Yaskawa INFORM job: A_ROOF_SIDE_0617_2_PAINT_45.JBI

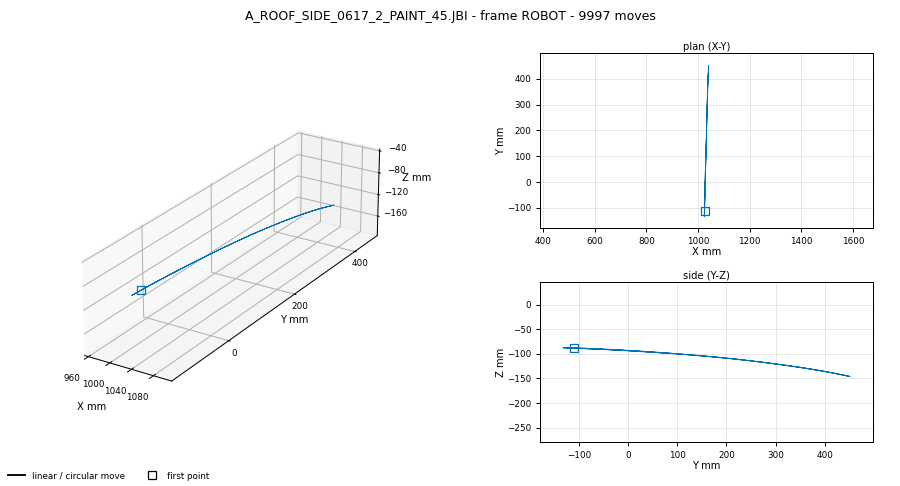
[picture p0: tool path of A_ROOF_SIDE_0617_2_PAINT_45.JBI in frame ROBOT, 9997 of 9997 moves have a stored position in this frame; points joined in program order, loops and branches not executed]
/JOB
//NAME A_ROOF_SIDE_0617_2_PAINT45
//POS
///NPOS 9997,0,0,0,0,0
///TOOL 1
///USER 0
///POSTYPE ROBOT
///RECTAN
///RCONF 1,0,0,0,0,0,0,0,0,0,0,0,0,0,0,0,0,0,0,0,0,0,0,0
C00000=1025.820,-110.808,-87.405,166.559,45.749,158.344
C00001=1025.826,-110.558,-87.414,166.562,45.746,158.343
C00002=1025.832,-110.309,-87.423,166.564,45.743,158.343
C00003=1025.837,-110.058,-87.432,166.568,45.740,158.343
C00004=1025.843,-109.809,-87.441,166.570,45.738,158.343
C00005=1025.849,-109.559,-87.450,166.574,45.735,158.343
C00006=1025.854,-109.310,-87.459,166.577,45.732,158.343
C00007=1025.860,-109.059,-87.468,166.579,45.729,158.343
C00008=1025.866,-108.810,-87.477,166.583,45.726,158.342
C00009=1025.872,-108.560,-87.486,166.586,45.724,158.342
C00010=1025.877,-108.311,-87.495,166.589,45.721,158.342
C00011=1025.883,-108.060,-87.504,166.592,45.718,158.342
C00012=1025.889,-107.811,-87.513,166.594,45.716,158.342
C00013=1025.895,-107.561,-87.522,166.598,45.713,158.342
C00014=1025.900,-107.312,-87.531,166.601,45.710,158.342
C00015=1025.906,-107.061,-87.540,166.604,45.708,158.341
C00016=1025.912,-106.812,-87.550,166.607,45.705,158.341
C00017=1025.918,-106.562,-87.558,166.609,45.703,158.341
C00018=1025.924,-106.312,-87.568,166.613,45.700,158.341
C00019=1025.929,-106.063,-87.577,166.616,45.697,158.341
C00020=1025.935,-105.812,-87.586,166.618,45.694,158.341
C00021=1025.941,-105.563,-87.595,166.622,45.692,158.341
C00022=1025.946,-105.313,-87.605,166.624,45.689,158.340
C00023=1025.952,-105.063,-87.614,166.628,45.686,158.340
C00024=1025.958,-104.814,-87.623,166.630,45.684,158.340
C00025=1025.964,-104.564,-87.633,166.634,45.681,158.340
C00026=1025.969,-104.314,-87.641,166.637,45.678,158.340
C00027=1025.975,-104.064,-87.651,166.640,45.676,158.340
C00028=1025.981,-103.814,-87.661,166.643,45.673,158.340
C00029=1025.986,-103.565,-87.670,166.645,45.670,158.340
C00030=1025.992,-103.315,-87.679,166.649,45.668,158.340
C00031=1025.998,-103.066,-87.688,166.651,45.665,158.339
C00032=1026.004,-102.816,-87.698,166.654,45.662,158.339
C00033=1026.010,-102.566,-87.707,166.658,45.659,158.339
C00034=1026.014,-102.316,-87.717,166.660,45.657,158.339
C00035=1026.021,-102.066,-87.726,166.664,45.654,158.339
C00036=1026.027,-101.817,-87.736,166.666,45.652,158.339
C00037=1026.032,-101.567,-87.745,166.670,45.649,158.339
C00038=1026.039,-101.281,-87.756,166.673,45.646,158.338
C00039=1026.046,-100.994,-87.767,166.676,45.643,158.338
C00040=1026.052,-100.708,-87.777,166.679,45.640,158.338
C00041=1026.059,-100.422,-87.789,166.683,45.637,158.338
C00042=1026.064,-100.173,-87.797,166.686,45.634,158.338
C00043=1026.070,-99.923,-87.807,166.690,45.631,158.338
C00044=1026.077,-99.673,-87.816,166.692,45.629,158.337
C00045=1026.083,-99.423,-87.826,166.696,45.626,158.337
C00046=1026.088,-99.174,-87.836,166.698,45.624,158.337
C00047=1026.094,-98.924,-87.845,166.701,45.621,158.337
C00048=1026.100,-98.674,-87.855,166.704,45.619,158.337
C00049=1026.106,-98.424,-87.864,166.707,45.616,158.337
C00050=1026.111,-98.175,-87.873,166.711,45.613,158.337
C00051=1026.117,-97.925,-87.883,166.713,45.610,158.336
C00052=1026.123,-97.675,-87.893,166.716,45.608,158.336
C00053=1026.129,-97.425,-87.902,166.719,45.605,158.336
C00054=1026.134,-97.176,-87.912,166.722,45.603,158.336
C00055=1026.140,-96.926,-87.922,166.725,45.600,158.336
C00056=1026.146,-96.676,-87.932,166.728,45.598,158.336
C00057=1026.152,-96.426,-87.941,166.731,45.595,158.336
C00058=1026.157,-96.176,-87.951,166.734,45.593,158.336
C00059=1026.163,-95.927,-87.961,166.737,45.590,158.336
C00060=1026.168,-95.677,-87.972,166.740,45.588,158.336
C00061=1026.175,-95.427,-87.981,166.742,45.585,158.335
C00062=1026.179,-95.178,-87.991,166.746,45.583,158.335
C00063=1026.186,-94.928,-88.001,166.748,45.580,158.335
C00064=1026.192,-94.678,-88.010,166.752,45.577,158.335
C00065=1026.197,-94.428,-88.020,166.754,45.575,158.335
C00066=1026.203,-94.178,-88.030,166.758,45.572,158.335
C00067=1026.208,-93.929,-88.040,166.760,45.570,158.335
C00068=1026.214,-93.679,-88.049,166.764,45.567,158.334
C00069=1026.220,-93.430,-88.060,166.766,45.565,158.334
C00070=1026.226,-93.180,-88.070,166.770,45.562,158.334
C00071=1026.232,-92.930,-88.080,166.772,45.560,158.334
C00072=1026.238,-92.680,-88.089,166.775,45.557,158.334
C00073=1026.243,-92.431,-88.099,166.778,45.555,158.334
C00074=1026.249,-92.182,-88.109,166.781,45.552,158.334
C00075=1026.255,-91.931,-88.120,166.785,45.550,158.334
C00076=1026.261,-91.682,-88.129,166.787,45.547,158.334
C00077=1026.266,-91.431,-88.139,166.791,45.545,158.334
C00078=1026.272,-91.182,-88.149,166.793,45.542,158.333
C00079=1026.278,-90.932,-88.160,166.797,45.539,158.333
C00080=1026.284,-90.682,-88.169,166.799,45.537,158.333
C00081=1026.289,-90.433,-88.179,166.802,45.534,158.333
C00082=1026.295,-90.183,-88.189,166.805,45.532,158.333
C00083=1026.301,-89.934,-88.200,166.808,45.529,158.333
C00084=1026.307,-89.684,-88.209,166.811,45.527,158.333
C00085=1026.313,-89.434,-88.219,166.814,45.524,158.332
C00086=1026.319,-89.185,-88.230,166.817,45.522,158.332
C00087=1026.325,-88.935,-88.240,166.820,45.519,158.332
C00088=1026.331,-88.685,-88.249,166.823,45.516,158.332
C00089=1026.336,-88.435,-88.260,166.826,45.514,158.332
C00090=1026.343,-88.185,-88.270,166.828,45.512,158.332
C00091=1026.348,-87.935,-88.280,166.832,45.509,158.332
C00092=1026.354,-87.686,-88.290,166.834,45.507,158.332
C00093=1026.360,-87.436,-88.300,166.838,45.504,158.332
C00094=1026.366,-87.186,-88.310,166.840,45.502,158.331
C00095=1026.372,-86.937,-88.321,166.844,45.499,158.331
C00096=1026.377,-86.687,-88.331,166.846,45.497,158.331
C00097=1026.384,-86.437,-88.341,166.850,45.494,158.331
C00098=1026.389,-86.187,-88.351,166.852,45.492,158.331
C00099=1026.395,-85.938,-88.361,166.856,45.489,158.331
C00100=1026.401,-85.688,-88.372,166.858,45.487,158.331
C00101=1026.407,-85.438,-88.381,166.861,45.484,158.330
C00102=1026.414,-85.154,-88.393,166.865,45.481,158.330
C00103=1026.420,-84.871,-88.404,166.868,45.478,158.330
C00104=1026.427,-84.586,-88.416,166.871,45.475,158.330
C00105=1026.434,-84.303,-88.428,166.875,45.472,158.330
C00106=1026.440,-84.053,-88.438,166.877,45.470,158.330
C00107=1026.445,-83.803,-88.449,166.881,45.467,158.330
C00108=1026.452,-83.554,-88.458,166.884,45.465,158.330
C00109=1026.458,-83.303,-88.469,166.887,45.462,158.329
C00110=1026.464,-83.054,-88.479,166.890,45.459,158.329
C00111=1026.470,-82.804,-88.490,166.893,45.457,158.329
C00112=1026.476,-82.554,-88.499,166.896,45.454,158.329
C00113=1026.482,-82.305,-88.510,166.899,45.452,158.329
C00114=1026.488,-82.055,-88.520,166.902,45.449,158.329
C00115=1026.494,-81.806,-88.531,166.904,45.446,158.328
C00116=1026.499,-81.556,-88.541,166.908,45.444,158.328
C00117=1026.506,-81.306,-88.551,166.910,45.441,158.328
C00118=1026.511,-81.056,-88.561,166.914,45.439,158.328
C00119=1026.518,-80.806,-88.572,166.916,45.436,158.328
C00120=1026.524,-80.557,-88.583,166.919,45.433,158.328
C00121=1026.530,-80.307,-88.592,166.922,45.431,158.328
C00122=1026.536,-80.058,-88.603,166.925,45.428,158.328
C00123=1026.541,-79.807,-88.614,166.928,45.426,158.327
C00124=1026.547,-79.558,-88.624,166.931,45.424,158.327
C00125=1026.553,-79.309,-88.635,166.934,45.421,158.327
C00126=1026.559,-79.058,-88.645,166.937,45.419,158.327
C00127=1026.565,-78.808,-88.656,166.940,45.417,158.327
C00128=1026.571,-78.559,-88.667,166.943,45.414,158.327
C00129=1026.577,-78.310,-88.678,166.946,45.412,158.327
C00130=1026.582,-78.059,-88.688,166.948,45.410,158.327
C00131=1026.589,-77.810,-88.698,166.952,45.407,158.326
C00132=1026.595,-77.560,-88.710,166.954,45.405,158.326
C00133=1026.601,-77.311,-88.720,166.958,45.402,158.326
C00134=1026.606,-77.061,-88.731,166.960,45.400,158.326
C00135=1026.612,-76.811,-88.741,166.963,45.397,158.326
C00136=1026.618,-76.561,-88.752,166.966,45.395,158.326
C00137=1026.624,-76.312,-88.763,166.970,45.392,158.326
C00138=1026.630,-76.062,-88.774,166.972,45.390,158.326
C00139=1026.636,-75.813,-88.785,166.976,45.387,158.326
C00140=1026.642,-75.562,-88.795,166.978,45.385,158.325
C00141=1026.647,-75.313,-88.806,166.980,45.383,158.325
C00142=1026.653,-75.064,-88.817,166.984,45.380,158.325
C00143=1026.660,-74.814,-88.827,166.986,45.378,158.325
C00144=1026.666,-74.564,-88.838,166.990,45.375,158.325
C00145=1026.672,-74.315,-88.849,166.992,45.373,158.325
C00146=1026.677,-74.065,-88.860,166.996,45.371,158.325
C00147=1026.684,-73.815,-88.871,166.998,45.368,158.325
C00148=1026.689,-73.565,-88.881,167.001,45.366,158.324
C00149=1026.694,-73.315,-88.893,167.004,45.364,158.324
C00150=1026.700,-73.066,-88.904,167.007,45.362,158.324
C00151=1026.706,-72.815,-88.915,167.009,45.359,158.324
C00152=1026.712,-72.566,-88.926,167.013,45.357,158.324
C00153=1026.718,-72.316,-88.937,167.016,45.355,158.324
C00154=1026.724,-72.068,-88.948,167.019,45.352,158.324
C00155=1026.730,-71.817,-88.960,167.021,45.350,158.324
C00156=1026.736,-71.568,-88.970,167.024,45.348,158.324
C00157=1026.741,-71.318,-88.982,167.028,45.345,158.324
C00158=1026.747,-71.068,-88.993,167.030,45.343,158.323
C00159=1026.753,-70.818,-89.004,167.033,45.341,158.323
C00160=1026.759,-70.569,-89.015,167.036,45.338,158.323
C00161=1026.764,-70.319,-89.026,167.039,45.336,158.323
C00162=1026.771,-70.069,-89.037,167.042,45.333,158.323
C00163=1026.776,-69.820,-89.048,167.045,45.331,158.323
C00164=1026.782,-69.570,-89.059,167.047,45.329,158.323
C00165=1026.788,-69.320,-89.071,167.051,45.326,158.323
C00166=1026.795,-69.039,-89.083,167.054,45.324,158.323
C00167=1026.801,-68.757,-89.096,167.056,45.322,158.323
C00168=1026.808,-68.475,-89.108,167.060,45.319,158.322
C00169=1026.814,-68.193,-89.121,167.063,45.316,158.322
C00170=1026.821,-67.944,-89.133,167.066,45.314,158.322
///RCONF 1,0,0,1,0,0,0,0,0,0,0,0,0,0,0,0,0,0,0,0,0,0,0,0
C00171=1026.827,-67.694,-89.143,167.069,45.311,158.322
C00172=1026.832,-67.445,-89.154,167.072,45.309,158.322
C00173=1026.838,-67.194,-89.166,167.075,45.307,158.322
C00174=1026.844,-66.945,-89.177,167.078,45.305,158.322
C00175=1026.850,-66.695,-89.189,167.080,45.302,158.322
C00176=1026.856,-66.445,-89.200,167.084,45.300,158.322
C00177=1026.862,-66.196,-89.211,167.087,45.298,158.322
C00178=1026.868,-65.946,-89.222,167.089,45.296,158.321
C00179=1026.874,-65.697,-89.234,167.093,45.293,158.321
C00180=1026.880,-65.446,-89.245,167.095,45.291,158.321
C00181=1026.885,-65.197,-89.256,167.097,45.289,158.321
C00182=1026.891,-64.947,-89.267,167.101,45.286,158.321
C00183=1026.898,-64.698,-89.279,167.104,45.284,158.321
C00184=1026.904,-64.448,-89.290,167.107,45.281,158.321
C00185=1026.910,-64.198,-89.301,167.110,45.279,158.321
C00186=1026.915,-63.949,-89.313,167.112,45.277,158.320
C00187=1026.922,-63.699,-89.325,167.116,45.274,158.320
C00188=1026.927,-63.449,-89.336,167.118,45.272,158.320
C00189=1026.933,-63.200,-89.347,167.121,45.270,158.320
C00190=1026.940,-62.950,-89.358,167.124,45.268,158.320
C00191=1026.945,-62.700,-89.370,167.127,45.266,158.320
C00192=1026.951,-62.451,-89.382,167.130,45.263,158.320
C00193=1026.957,-62.201,-89.393,167.133,45.261,158.320
C00194=1026.963,-61.951,-89.404,167.135,45.259,158.320
C00195=1026.969,-61.702,-89.416,167.138,45.256,158.319
C00196=1026.976,-61.452,-89.427,167.141,45.254,158.319
C00197=1026.981,-61.202,-89.438,167.144,45.252,158.319
C00198=1026.987,-60.953,-89.450,167.147,45.249,158.319
C00199=1026.993,-60.703,-89.461,167.150,45.247,158.319
C00200=1027.000,-60.454,-89.473,167.152,45.245,158.319
C00201=1027.006,-60.204,-89.484,167.156,45.242,158.319
C00202=1027.011,-59.954,-89.497,167.158,45.240,158.319
C00203=1027.018,-59.704,-89.508,167.162,45.238,158.319
C00204=1027.024,-59.455,-89.519,167.164,45.235,158.318
C00205=1027.030,-59.205,-89.531,167.167,45.233,158.318
C00206=1027.036,-58.956,-89.541,167.170,45.230,158.318
C00207=1027.042,-58.706,-89.554,167.173,45.228,158.318
C00208=1027.048,-58.456,-89.565,167.175,45.226,158.318
C00209=1027.054,-58.207,-89.577,167.178,45.223,158.318
C00210=1027.061,-57.956,-89.588,167.181,45.221,158.318
C00211=1027.066,-57.707,-89.600,167.185,45.219,158.318
C00212=1027.072,-57.457,-89.612,167.187,45.216,158.317
C00213=1027.078,-57.208,-89.623,167.190,45.214,158.317
C00214=1027.085,-56.958,-89.634,167.193,45.211,158.317
C00215=1027.091,-56.708,-89.646,167.195,45.209,158.317
C00216=1027.097,-56.459,-89.659,167.198,45.207,158.317
C00217=1027.103,-56.209,-89.670,167.201,45.204,158.317
C00218=1027.109,-55.960,-89.681,167.204,45.202,158.317
C00219=1027.115,-55.710,-89.693,167.207,45.199,158.316
C00220=1027.122,-55.460,-89.705,167.210,45.197,158.316
C00221=1027.127,-55.211,-89.716,167.213,45.195,158.316
C00222=1027.134,-54.961,-89.728,167.216,45.192,158.316
C00223=1027.140,-54.712,-89.740,167.218,45.190,158.316
C00224=1027.146,-54.462,-89.751,167.221,45.188,158.316
C00225=1027.152,-54.212,-89.763,167.224,45.185,158.316
C00226=1027.158,-53.962,-89.775,167.227,45.183,158.316
C00227=1027.164,-53.713,-89.786,167.229,45.181,158.315
C00228=1027.171,-53.464,-89.798,167.233,45.179,158.315
C00229=1027.177,-53.213,-89.810,167.235,45.176,158.315
C00230=1027.183,-52.933,-89.823,167.239,45.174,158.315
C00231=1027.191,-52.652,-89.836,167.242,45.171,158.315
C00232=1027.197,-52.372,-89.850,167.246,45.168,158.315
C00233=1027.205,-52.091,-89.863,167.248,45.165,158.315
C00234=1027.211,-51.842,-89.874,167.252,45.163,158.314
C00235=1027.217,-51.592,-89.886,167.254,45.160,158.314
C00236=1027.223,-51.342,-89.899,167.256,45.158,158.314
C00237=1027.230,-51.092,-89.910,167.260,45.156,158.314
C00238=1027.236,-50.843,-89.922,167.262,45.153,158.314
C00239=1027.241,-50.593,-89.934,167.266,45.151,158.314
C00240=1027.248,-50.344,-89.946,167.269,45.149,158.314
C00241=1027.254,-50.093,-89.958,167.271,45.146,158.314
C00242=1027.259,-49.844,-89.970,167.273,45.144,158.313
C00243=1027.266,-49.594,-89.982,167.277,45.142,158.313
C00244=1027.272,-49.345,-89.995,167.280,45.140,158.313
C00245=1027.278,-49.095,-90.007,167.282,45.138,158.313
C00246=1027.284,-48.846,-90.019,167.285,45.136,158.313
C00247=1027.289,-48.596,-90.031,167.288,45.133,158.313
C00248=1027.296,-48.346,-90.043,167.291,45.131,158.313
C00249=1027.302,-48.096,-90.056,167.293,45.129,158.313
C00250=1027.308,-47.848,-90.067,167.296,45.127,158.313
C00251=1027.314,-47.598,-90.080,167.299,45.125,158.313
C00252=1027.320,-47.348,-90.093,167.302,45.122,158.312
C00253=1027.326,-47.098,-90.105,167.304,45.120,158.312
C00254=1027.332,-46.849,-90.117,167.307,45.118,158.312
C00255=1027.338,-46.599,-90.129,167.311,45.116,158.312
C00256=1027.344,-46.350,-90.141,167.313,45.113,158.312
C00257=1027.350,-46.100,-90.154,167.316,45.111,158.312
C00258=1027.356,-45.850,-90.166,167.319,45.109,158.312
C00259=1027.362,-45.601,-90.178,167.322,45.107,158.312
C00260=1027.368,-45.351,-90.191,167.324,45.105,158.312
C00261=1027.375,-45.102,-90.202,167.327,45.103,158.311
C00262=1027.381,-44.852,-90.215,167.330,45.100,158.311
C00263=1027.387,-44.602,-90.228,167.333,45.098,158.311
C00264=1027.393,-44.352,-90.240,167.335,45.096,158.311
C00265=1027.399,-44.103,-90.252,167.338,45.094,158.311
C00266=1027.404,-43.853,-90.264,167.341,45.091,158.311
C00267=1027.411,-43.604,-90.276,167.344,45.089,158.311
C00268=1027.417,-43.354,-90.289,167.346,45.087,158.311
C00269=1027.423,-43.104,-90.301,167.349,45.085,158.310
C00270=1027.430,-42.854,-90.313,167.352,45.083,158.310
C00271=1027.436,-42.605,-90.327,167.355,45.081,158.310
C00272=1027.441,-42.356,-90.339,167.358,45.079,158.310
C00273=1027.448,-42.106,-90.351,167.360,45.076,158.310
C00274=1027.454,-41.856,-90.363,167.364,45.074,158.310
C00275=1027.460,-41.606,-90.376,167.366,45.072,158.310
C00276=1027.466,-41.357,-90.388,167.369,45.070,158.310
C00277=1027.472,-41.107,-90.400,167.371,45.067,158.309
C00278=1027.478,-40.858,-90.414,167.375,45.065,158.309
C00279=1027.485,-40.608,-90.426,167.377,45.063,158.309
C00280=1027.491,-40.358,-90.438,167.380,45.061,158.309
C00281=1027.497,-40.108,-90.451,167.382,45.058,158.309
C00282=1027.503,-39.859,-90.463,167.386,45.056,158.309
C00283=1027.509,-39.610,-90.476,167.388,45.054,158.309
C00284=1027.515,-39.360,-90.488,167.391,45.051,158.309
C00285=1027.522,-39.111,-90.500,167.394,45.049,158.309
C00286=1027.528,-38.861,-90.513,167.397,45.047,158.308
C00287=1027.534,-38.612,-90.526,167.399,45.045,158.308
C00288=1027.540,-38.362,-90.538,167.402,45.043,158.308
C00289=1027.546,-38.112,-90.551,167.405,45.041,158.308
C00290=1027.551,-37.862,-90.564,167.408,45.038,158.308
C00291=1027.558,-37.613,-90.577,167.411,45.036,158.308
C00292=1027.564,-37.363,-90.589,167.413,45.034,158.308
C00293=1027.570,-37.114,-90.603,167.416,45.032,158.308
C00294=1027.577,-36.833,-90.617,167.419,45.030,158.308
C00295=1027.584,-36.553,-90.631,167.422,45.027,158.307
C00296=1027.590,-36.273,-90.645,167.425,45.025,158.307
C00297=1027.597,-35.993,-90.660,167.428,45.023,158.307
C00298=1027.603,-35.743,-90.673,167.431,45.020,158.307
C00299=1027.610,-35.494,-90.685,167.434,45.018,158.307
C00300=1027.616,-35.244,-90.698,167.436,45.016,158.307
C00301=1027.622,-34.994,-90.710,167.439,45.014,158.307
C00302=1027.628,-34.745,-90.724,167.442,45.012,158.307
C00303=1027.634,-34.495,-90.736,167.445,45.010,158.307
C00304=1027.640,-34.246,-90.749,167.447,45.007,158.306
C00305=1027.646,-33.996,-90.762,167.450,45.005,158.306
C00306=1027.652,-33.747,-90.775,167.453,45.003,158.306
C00307=1027.658,-33.497,-90.788,167.455,45.001,158.306
C00308=1027.664,-33.247,-90.801,167.458,44.999,158.306
C00309=1027.670,-32.998,-90.814,167.461,44.997,158.306
C00310=1027.676,-32.748,-90.827,167.464,44.995,158.306
C00311=1027.682,-32.498,-90.839,167.466,44.993,158.306
C00312=1027.688,-32.249,-90.853,167.469,44.991,158.306
C00313=1027.695,-31.999,-90.866,167.471,44.989,158.305
C00314=1027.701,-31.749,-90.879,167.475,44.986,158.305
C00315=1027.707,-31.499,-90.891,167.477,44.984,158.305
C00316=1027.713,-31.250,-90.905,167.480,44.982,158.305
C00317=1027.719,-31.001,-90.918,167.483,44.980,158.305
C00318=1027.726,-30.751,-90.930,167.485,44.978,158.305
C00319=1027.732,-30.502,-90.943,167.489,44.976,158.305
C00320=1027.738,-30.252,-90.956,167.491,44.973,158.305
C00321=1027.744,-30.003,-90.969,167.494,44.971,158.304
C00322=1027.750,-29.753,-90.982,167.496,44.969,158.304
C00323=1027.757,-29.503,-90.995,167.499,44.967,158.304
C00324=1027.763,-29.254,-91.008,167.501,44.965,158.304
C00325=1027.769,-29.004,-91.021,167.505,44.962,158.304
C00326=1027.775,-28.755,-91.034,167.507,44.960,158.304
C00327=1027.782,-28.505,-91.048,167.510,44.958,158.304
C00328=1027.788,-28.255,-91.060,167.513,44.956,158.304
C00329=1027.794,-28.006,-91.073,167.515,44.953,158.303
C00330=1027.801,-27.756,-91.087,167.518,44.951,158.303
C00331=1027.806,-27.506,-91.100,167.521,44.949,158.303
C00332=1027.813,-27.257,-91.113,167.524,44.947,158.303
C00333=1027.819,-27.008,-91.126,167.526,44.945,158.303
C00334=1027.824,-26.758,-91.139,167.529,44.943,158.303
C00335=1027.830,-26.508,-91.153,167.531,44.941,158.303
C00336=1027.837,-26.258,-91.166,167.534,44.939,158.303
C00337=1027.843,-26.009,-91.179,167.536,44.937,158.303
C00338=1027.849,-25.760,-91.193,167.540,44.934,158.302
C00339=1027.855,-25.510,-91.206,167.543,44.932,158.302
C00340=1027.861,-25.260,-91.219,167.545,44.930,158.302
///RCONF 1,0,0,0,0,0,0,0,0,0,0,0,0,0,0,0,0,0,0,0,0,0,0,0
C00341=1027.867,-25.011,-91.232,167.548,44.928,158.302
C00342=1027.873,-24.761,-91.247,167.550,44.926,158.302
C00343=1027.879,-24.512,-91.260,167.553,44.925,158.302
C00344=1027.886,-24.262,-91.273,167.555,44.923,158.302
C00345=1027.892,-24.012,-91.286,167.558,44.921,158.302
C00346=1027.897,-23.763,-91.300,167.561,44.919,158.302
C00347=1027.904,-23.513,-91.313,167.564,44.916,158.302
C00348=1027.910,-23.264,-91.326,167.567,44.914,158.301
C00349=1027.916,-23.014,-91.340,167.569,44.912,158.301
C00350=1027.922,-22.765,-91.354,167.572,44.910,158.301
C00351=1027.928,-22.516,-91.367,167.574,44.908,158.301
C00352=1027.935,-22.266,-91.381,167.577,44.906,158.301
C00353=1027.941,-22.016,-91.394,167.579,44.904,158.301
C00354=1027.946,-21.767,-91.408,167.582,44.902,158.301
C00355=1027.953,-21.518,-91.421,167.585,44.900,158.301
C00356=1027.959,-21.267,-91.434,167.588,44.898,158.301
C00357=1027.965,-21.018,-91.447,167.591,44.895,158.300
C00358=1027.972,-20.737,-91.463,167.593,44.893,158.300
C00359=1027.979,-20.455,-91.479,167.597,44.891,158.300
C00360=1027.986,-20.175,-91.493,167.599,44.888,158.300
C00361=1027.993,-19.894,-91.508,167.603,44.886,158.300
C00362=1027.999,-19.644,-91.522,167.605,44.884,158.300
C00363=1028.006,-19.394,-91.535,167.608,44.881,158.300
C00364=1028.011,-19.145,-91.549,167.610,44.879,158.299
C00365=1028.018,-18.896,-91.562,167.613,44.877,158.299
C00366=1028.024,-18.646,-91.576,167.615,44.875,158.299
C00367=1028.030,-18.396,-91.590,167.618,44.873,158.299
C00368=1028.036,-18.147,-91.603,167.622,44.871,158.299
C00369=1028.043,-17.897,-91.617,167.624,44.869,158.299
C00370=1028.049,-17.648,-91.630,167.627,44.867,158.299
C00371=1028.055,-17.398,-91.644,167.629,44.865,158.299
C00372=1028.061,-17.148,-91.658,167.632,44.863,158.298
C00373=1028.068,-16.899,-91.672,167.634,44.861,158.298
C00374=1028.073,-16.650,-91.685,167.637,44.859,158.298
C00375=1028.080,-16.400,-91.699,167.639,44.856,158.298
C00376=1028.087,-16.151,-91.712,167.642,44.854,158.298
C00377=1028.093,-15.901,-91.726,167.645,44.852,158.298
C00378=1028.099,-15.651,-91.740,167.648,44.850,158.298
C00379=1028.105,-15.402,-91.753,167.651,44.848,158.298
C00380=1028.111,-15.151,-91.767,167.653,44.846,158.298
C00381=1028.118,-14.903,-91.781,167.656,44.844,158.297
C00382=1028.123,-14.653,-91.795,167.658,44.842,158.297
C00383=1028.130,-14.403,-91.809,167.661,44.840,158.297
C00384=1028.135,-14.154,-91.823,167.663,44.838,158.297
C00385=1028.142,-13.904,-91.836,167.666,44.836,158.297
C00386=1028.148,-13.655,-91.851,167.669,44.834,158.297
C00387=1028.153,-13.405,-91.865,167.671,44.832,158.297
C00388=1028.160,-13.155,-91.878,167.674,44.829,158.297
C00389=1028.166,-12.906,-91.893,167.676,44.827,158.296
C00390=1028.172,-12.657,-91.906,167.679,44.825,158.296
C00391=1028.178,-12.407,-91.921,167.681,44.824,158.296
C00392=1028.185,-12.157,-91.934,167.684,44.822,158.296
C00393=1028.191,-11.908,-91.949,167.687,44.820,158.296
C00394=1028.197,-11.659,-91.962,167.689,44.818,158.296
C00395=1028.203,-11.408,-91.976,167.692,44.816,158.296
C00396=1028.210,-11.160,-91.990,167.694,44.814,158.296
C00397=1028.215,-10.910,-92.004,167.697,44.812,158.296
C00398=1028.221,-10.660,-92.018,167.699,44.810,158.295
C00399=1028.228,-10.411,-92.032,167.703,44.808,158.295
C00400=1028.234,-10.161,-92.047,167.706,44.806,158.295
C00401=1028.240,-9.912,-92.061,167.708,44.804,158.295
C00402=1028.247,-9.662,-92.075,167.711,44.801,158.295
C00403=1028.253,-9.413,-92.088,167.713,44.799,158.295
C00404=1028.259,-9.163,-92.103,167.716,44.797,158.295
C00405=1028.265,-8.913,-92.117,167.718,44.795,158.295
C00406=1028.271,-8.663,-92.130,167.721,44.793,158.295
C00407=1028.277,-8.415,-92.145,167.723,44.791,158.294
C00408=1028.284,-8.165,-92.159,167.726,44.789,158.294
C00409=1028.290,-7.916,-92.173,167.729,44.787,158.294
C00410=1028.297,-7.666,-92.187,167.731,44.785,158.294
C00411=1028.302,-7.417,-92.201,167.734,44.783,158.294
C00412=1028.308,-7.166,-92.216,167.736,44.781,158.294
C00413=1028.315,-6.918,-92.230,167.739,44.779,158.294
C00414=1028.321,-6.667,-92.244,167.741,44.777,158.294
C00415=1028.327,-6.418,-92.257,167.744,44.775,158.293
C00416=1028.334,-6.169,-92.272,167.747,44.773,158.293
C00417=1028.340,-5.919,-92.285,167.749,44.771,158.293
C00418=1028.346,-5.670,-92.300,167.751,44.768,158.293
C00419=1028.352,-5.420,-92.314,167.754,44.766,158.293
C00420=1028.359,-5.171,-92.329,167.757,44.764,158.293
C00421=1028.364,-4.921,-92.342,167.759,44.762,158.293
C00422=1028.372,-4.639,-92.359,167.763,44.760,158.293
C00423=1028.379,-4.356,-92.375,167.765,44.757,158.292
C00424=1028.386,-4.072,-92.391,167.769,44.755,158.292
C00425=1028.394,-3.791,-92.407,167.771,44.752,158.292
C00426=1028.399,-3.542,-92.422,167.774,44.751,158.292
C00427=1028.405,-3.291,-92.436,167.776,44.749,158.292
C00428=1028.412,-3.042,-92.451,167.779,44.747,158.292
C00429=1028.418,-2.793,-92.466,167.782,44.745,158.292
C00430=1028.424,-2.542,-92.480,167.784,44.743,158.292
C00431=1028.429,-2.293,-92.494,167.787,44.741,158.291
C00432=1028.436,-2.044,-92.509,167.789,44.739,158.291
C00433=1028.441,-1.794,-92.523,167.792,44.737,158.291
C00434=1028.448,-1.545,-92.538,167.795,44.735,158.291
C00435=1028.454,-1.296,-92.552,167.797,44.734,158.291
C00436=1028.461,-1.046,-92.567,167.800,44.732,158.291
C00437=1028.467,-0.796,-92.581,167.802,44.730,158.291
C00438=1028.472,-0.547,-92.596,167.805,44.728,158.291
C00439=1028.479,-0.297,-92.611,167.808,44.726,158.291
C00440=1028.485,-0.048,-92.626,167.810,44.724,158.290
C00441=1028.491,0.202,-92.640,167.812,44.722,158.290
C00442=1028.497,0.452,-92.655,167.814,44.720,158.290
C00443=1028.503,0.700,-92.669,167.817,44.718,158.290
C00444=1028.509,0.950,-92.684,167.819,44.716,158.290
C00445=1028.516,1.200,-92.699,167.822,44.714,158.290
C00446=1028.521,1.449,-92.713,167.825,44.712,158.290
C00447=1028.527,1.699,-92.728,167.827,44.710,158.290
C00448=1028.533,1.948,-92.743,167.830,44.708,158.290
C00449=1028.540,2.198,-92.757,167.832,44.706,158.289
C00450=1028.546,2.447,-92.772,167.835,44.704,158.289
C00451=1028.553,2.696,-92.786,167.838,44.702,158.289
C00452=1028.559,2.946,-92.801,167.840,44.700,158.289
C00453=1028.565,3.196,-92.816,167.843,44.698,158.289
C00454=1028.571,3.445,-92.830,167.845,44.696,158.289
C00455=1028.577,3.694,-92.845,167.848,44.694,158.289
C00456=1028.584,3.944,-92.860,167.851,44.692,158.289
C00457=1028.589,4.193,-92.875,167.853,44.691,158.289
C00458=1028.596,4.443,-92.890,167.855,44.688,158.288
C00459=1028.602,4.692,-92.905,167.858,44.686,158.288
C00460=1028.608,4.942,-92.919,167.861,44.684,158.288
C00461=1028.614,5.192,-92.933,167.863,44.682,158.288
C00462=1028.620,5.441,-92.948,167.866,44.680,158.288
C00463=1028.627,5.691,-92.963,167.868,44.678,158.288
C00464=1028.632,5.940,-92.978,167.870,44.676,158.288
C00465=1028.639,6.190,-92.993,167.873,44.674,158.287
C00466=1028.645,6.439,-93.008,167.875,44.672,158.287
C00467=1028.652,6.689,-93.023,167.878,44.670,158.287
C00468=1028.657,6.938,-93.037,167.880,44.668,158.287
C00469=1028.664,7.187,-93.052,167.883,44.667,158.287
C00470=1028.670,7.427,-93.067,167.885,44.665,158.287
C00471=1028.676,7.667,-93.080,167.888,44.663,158.287
C00472=1028.682,7.907,-93.095,167.891,44.661,158.287
C00473=1028.688,8.147,-93.109,167.893,44.659,158.286
C00474=1028.694,8.387,-93.124,167.896,44.657,158.286
C00475=1028.700,8.626,-93.138,167.897,44.655,158.286
C00476=1028.706,8.866,-93.152,167.900,44.653,158.286
C00477=1028.713,9.106,-93.167,167.903,44.651,158.286
C00478=1028.718,9.355,-93.181,167.905,44.648,158.286
C00479=1028.725,9.605,-93.196,167.908,44.646,158.286
C00480=1028.731,9.855,-93.211,167.910,44.644,158.285
C00481=1028.738,10.104,-93.226,167.913,44.643,158.285
C00482=1028.744,10.354,-93.241,167.915,44.641,158.285
C00483=1028.750,10.603,-93.256,167.918,44.639,158.285
C00484=1028.756,10.853,-93.271,167.920,44.637,158.285
C00485=1028.762,11.102,-93.286,167.923,44.635,158.285
C00486=1028.771,11.406,-93.304,167.925,44.632,158.285
C00487=1028.778,11.709,-93.322,167.929,44.629,158.284
C00488=1028.786,12.014,-93.340,167.932,44.627,158.284
C00489=1028.793,12.317,-93.358,167.935,44.624,158.284
C00490=1028.800,12.567,-93.373,167.937,44.622,158.284
C00491=1028.806,12.817,-93.388,167.940,44.621,158.284
C00492=1028.813,13.066,-93.404,167.942,44.619,158.284
C00493=1028.819,13.315,-93.419,167.945,44.616,158.284
C00494=1028.826,13.565,-93.434,167.947,44.614,158.283
C00495=1028.832,13.815,-93.449,167.950,44.612,158.283
C00496=1028.837,14.064,-93.464,167.953,44.610,158.283
C00497=1028.844,14.313,-93.480,167.955,44.608,158.283
C00498=1028.850,14.563,-93.494,167.958,44.606,158.283
C00499=1028.856,14.812,-93.509,167.960,44.604,158.283
C00500=1028.862,15.062,-93.525,167.962,44.602,158.283
C00501=1028.869,15.311,-93.541,167.965,44.601,158.283
C00502=1028.875,15.561,-93.556,167.967,44.599,158.282
C00503=1028.881,15.811,-93.571,167.970,44.597,158.282
C00504=1028.887,16.059,-93.586,167.972,44.595,158.282
C00505=1028.893,16.309,-93.601,167.975,44.593,158.282
C00506=1028.900,16.558,-93.616,167.977,44.591,158.282
C00507=1028.906,16.808,-93.633,167.980,44.589,158.282
C00508=1028.912,17.058,-93.647,167.983,44.587,158.282
C00509=1028.918,17.307,-93.662,167.985,44.585,158.282
C00510=1028.925,17.556,-93.678,167.987,44.583,158.281
C00511=1028.931,17.806,-93.694,167.989,44.581,158.281
C00512=1028.937,18.055,-93.709,167.992,44.579,158.281
C00513=1028.943,18.304,-93.724,167.995,44.577,158.281
C00514=1028.949,18.554,-93.739,167.997,44.575,158.281
C00515=1028.956,18.803,-93.755,168.000,44.573,158.281
C00516=1028.962,19.053,-93.770,168.002,44.571,158.281
C00517=1028.968,19.302,-93.785,168.005,44.569,158.280
C00518=1028.974,19.552,-93.801,168.007,44.567,158.280
C00519=1028.981,19.801,-93.816,168.009,44.565,158.280
C00520=1028.987,20.051,-93.832,168.011,44.563,158.280
C00521=1028.993,20.300,-93.847,168.014,44.561,158.280
C00522=1029.000,20.550,-93.863,168.017,44.559,158.280
C00523=1029.005,20.799,-93.879,168.019,44.557,158.280
C00524=1029.012,21.049,-93.894,168.022,44.555,158.280
C00525=1029.018,21.299,-93.910,168.024,44.553,158.279
C00526=1029.024,21.548,-93.925,168.027,44.551,158.279
C00527=1029.030,21.798,-93.941,168.029,44.550,158.279
C00528=1029.037,22.047,-93.957,168.031,44.548,158.279
C00529=1029.043,22.296,-93.972,168.034,44.546,158.279
C00530=1029.049,22.546,-93.988,168.036,44.544,158.279
C00531=1029.056,22.795,-94.004,168.039,44.542,158.279
C00532=1029.061,23.045,-94.019,168.041,44.540,158.279
C00533=1029.068,23.294,-94.035,168.044,44.538,158.278
C00534=1029.074,23.544,-94.050,168.047,44.536,158.278
C00535=1029.080,23.793,-94.066,168.048,44.534,158.278
C00536=1029.087,24.042,-94.081,168.051,44.532,158.278
C00537=1029.093,24.292,-94.097,168.053,44.530,158.278
C00538=1029.099,24.541,-94.113,168.056,44.528,158.278
C00539=1029.105,24.791,-94.128,168.059,44.527,158.278
C00540=1029.112,25.040,-94.144,168.061,44.525,158.278
C00541=1029.117,25.290,-94.160,168.064,44.523,158.277
C00542=1029.124,25.539,-94.175,168.066,44.521,158.277
C00543=1029.131,25.788,-94.191,168.068,44.518,158.277
C00544=1029.136,26.038,-94.206,168.070,44.516,158.277
C00545=1029.143,26.287,-94.222,168.073,44.514,158.277
C00546=1029.149,26.536,-94.238,168.075,44.512,158.277
C00547=1029.155,26.786,-94.253,168.078,44.510,158.277
C00548=1029.161,27.035,-94.270,168.081,44.509,158.276
C00549=1029.167,27.284,-94.286,168.083,44.507,158.276
C00550=1029.175,27.570,-94.304,168.086,44.505,158.276
C00551=1029.182,27.856,-94.321,168.088,44.502,158.276
C00552=1029.189,28.142,-94.340,168.092,44.500,158.276
C00553=1029.196,28.428,-94.358,168.094,44.498,158.276
C00554=1029.203,28.677,-94.374,168.097,44.496,158.276
C00555=1029.208,28.927,-94.389,168.099,44.494,158.275
C00556=1029.214,29.177,-94.406,168.101,44.492,158.275
C00557=1029.221,29.426,-94.421,168.104,44.490,158.275
C00558=1029.227,29.675,-94.438,168.106,44.488,158.275
C00559=1029.233,29.924,-94.454,168.109,44.486,158.275
C00560=1029.240,30.173,-94.470,168.112,44.485,158.275
C00561=1029.245,30.423,-94.485,168.113,44.483,158.275
C00562=1029.251,30.673,-94.501,168.116,44.481,158.275
C00563=1029.259,30.922,-94.517,168.118,44.479,158.274
C00564=1029.265,31.172,-94.534,168.121,44.477,158.274
C00565=1029.270,31.421,-94.550,168.123,44.475,158.274
C00566=1029.277,31.670,-94.566,168.126,44.473,158.274
C00567=1029.283,31.920,-94.582,168.128,44.471,158.274
C00568=1029.289,32.169,-94.598,168.130,44.469,158.274
C00569=1029.295,32.419,-94.614,168.133,44.467,158.274
C00570=1029.301,32.668,-94.629,168.135,44.466,158.274
C00571=1029.308,32.918,-94.646,168.138,44.464,158.273
C00572=1029.314,33.167,-94.662,168.141,44.462,158.273
C00573=1029.321,33.416,-94.678,168.142,44.460,158.273
C00574=1029.327,33.666,-94.694,168.145,44.458,158.273
C00575=1029.332,33.915,-94.710,168.147,44.456,158.273
C00576=1029.339,34.164,-94.726,168.150,44.454,158.273
C00577=1029.345,34.413,-94.742,168.153,44.452,158.273
C00578=1029.352,34.663,-94.759,168.155,44.450,158.272
C00579=1029.358,34.913,-94.775,168.158,44.448,158.272
C00580=1029.364,35.162,-94.791,168.159,44.447,158.272
C00581=1029.370,35.411,-94.807,168.162,44.444,158.272
C00582=1029.376,35.661,-94.823,168.164,44.442,158.272
C00583=1029.384,35.910,-94.839,168.167,44.440,158.272
C00584=1029.389,36.160,-94.856,168.169,44.438,158.272
C00585=1029.395,36.409,-94.872,168.172,44.436,158.271
C00586=1029.402,36.658,-94.888,168.174,44.434,158.271
C00587=1029.408,36.907,-94.904,168.176,44.432,158.271
C00588=1029.415,37.157,-94.920,168.179,44.431,158.271
C00589=1029.421,37.407,-94.937,168.181,44.429,158.271
C00590=1029.427,37.656,-94.953,168.184,44.427,158.271
C00591=1029.432,37.905,-94.969,168.187,44.425,158.271
C00592=1029.438,38.155,-94.985,168.188,44.423,158.270
C00593=1029.445,38.405,-95.002,168.191,44.421,158.270
C00594=1029.451,38.654,-95.018,168.193,44.419,158.270
C00595=1029.458,38.903,-95.035,168.196,44.417,158.270
C00596=1029.464,39.152,-95.051,168.198,44.415,158.270
C00597=1029.470,39.401,-95.067,168.200,44.414,158.270
C00598=1029.476,39.651,-95.084,168.203,44.412,158.270
C00599=1029.482,39.901,-95.100,168.205,44.410,158.270
C00600=1029.488,40.150,-95.116,168.208,44.408,158.269
C00601=1029.495,40.399,-95.133,168.210,44.406,158.269
C00602=1029.501,40.649,-95.150,168.212,44.404,158.269
C00603=1029.507,40.898,-95.166,168.215,44.402,158.269
C00604=1029.513,41.148,-95.182,168.217,44.400,158.269
C00605=1029.519,41.397,-95.199,168.220,44.398,158.269
C00606=1029.526,41.646,-95.216,168.222,44.396,158.269
C00607=1029.532,41.896,-95.232,168.224,44.395,158.268
C00608=1029.538,42.145,-95.249,168.226,44.393,158.268
C00609=1029.544,42.394,-95.265,168.229,44.391,158.268
C00610=1029.550,42.644,-95.282,168.232,44.389,158.268
C00611=1029.556,42.893,-95.298,168.234,44.387,158.268
C00612=1029.562,43.142,-95.315,168.236,44.386,158.268
C00613=1029.569,43.391,-95.332,168.239,44.384,158.268
C00614=1029.575,43.678,-95.351,168.241,44.382,158.268
C00615=1029.583,43.964,-95.370,168.244,44.379,158.267
C00616=1029.589,44.249,-95.389,168.247,44.377,158.267
C00617=1029.596,44.535,-95.408,168.250,44.375,158.267
C00618=1029.603,44.784,-95.425,168.252,44.373,158.267
C00619=1029.609,45.035,-95.442,168.254,44.372,158.267
C00620=1029.615,45.283,-95.459,168.257,44.370,158.267
C00621=1029.621,45.533,-95.475,168.259,44.368,158.267
C00622=1029.628,45.782,-95.493,168.262,44.366,158.267
C00623=1029.633,46.032,-95.509,168.264,44.365,158.266
C00624=1029.639,46.281,-95.526,168.266,44.363,158.266
C00625=1029.645,46.530,-95.543,168.269,44.361,158.266
C00626=1029.652,46.780,-95.559,168.271,44.359,158.266
C00627=1029.658,47.029,-95.576,168.273,44.357,158.266
C00628=1029.663,47.278,-95.593,168.276,44.355,158.266
C00629=1029.670,47.528,-95.610,168.278,44.353,158.266
C00630=1029.676,47.777,-95.627,168.281,44.352,158.266
C00631=1029.682,48.026,-95.644,168.283,44.350,158.266
C00632=1029.688,48.276,-95.661,168.285,44.348,158.265
C00633=1029.694,48.525,-95.678,168.288,44.346,158.265
C00634=1029.700,48.774,-95.694,168.290,44.345,158.265
C00635=1029.707,49.024,-95.711,168.292,44.343,158.265
C00636=1029.712,49.273,-95.728,168.294,44.341,158.265
C00637=1029.718,49.522,-95.745,168.297,44.339,158.265
C00638=1029.725,49.772,-95.762,168.300,44.337,158.265
C00639=1029.731,50.021,-95.779,168.302,44.335,158.264
C00640=1029.736,50.270,-95.796,168.304,44.333,158.264
C00641=1029.743,50.520,-95.813,168.306,44.331,158.264
C00642=1029.749,50.769,-95.829,168.309,44.329,158.264
C00643=1029.756,51.019,-95.847,168.312,44.328,158.264
C00644=1029.762,51.268,-95.863,168.313,44.326,158.264
C00645=1029.768,51.517,-95.880,168.316,44.324,158.264
C00646=1029.774,51.766,-95.898,168.318,44.322,158.263
C00647=1029.780,52.016,-95.914,168.321,44.320,158.263
C00648=1029.787,52.265,-95.931,168.323,44.318,158.263
C00649=1029.793,52.515,-95.948,168.325,44.316,158.263
C00650=1029.799,52.764,-95.965,168.328,44.314,158.263
C00651=1029.806,53.013,-95.982,168.330,44.313,158.263
C00652=1029.811,53.263,-95.999,168.333,44.311,158.263
C00653=1029.818,53.512,-96.017,168.335,44.310,158.263
C00654=1029.824,53.761,-96.034,168.337,44.308,158.263
C00655=1029.831,54.011,-96.050,168.340,44.306,158.262
C00656=1029.836,54.260,-96.068,168.343,44.304,158.262
C00657=1029.842,54.509,-96.084,168.345,44.302,158.262
C00658=1029.849,54.759,-96.101,168.346,44.299,158.262
C00659=1029.855,55.007,-96.118,168.349,44.298,158.262
C00660=1029.861,55.258,-96.136,168.352,44.296,158.262
C00661=1029.867,55.507,-96.153,168.354,44.294,158.261
C00662=1029.874,55.756,-96.170,168.356,44.292,158.261
C00663=1029.880,56.005,-96.187,168.358,44.290,158.261
C00664=1029.886,56.255,-96.204,168.361,44.288,158.261
C00665=1029.892,56.504,-96.221,168.364,44.286,158.261
C00666=1029.899,56.753,-96.238,168.366,44.284,158.261
C00667=1029.905,57.003,-96.255,168.368,44.283,158.261
C00668=1029.911,57.252,-96.273,168.370,44.281,158.260
C00669=1029.918,57.501,-96.290,168.373,44.279,158.260
C00670=1029.924,57.750,-96.307,168.376,44.277,158.260
C00671=1029.930,58.000,-96.324,168.378,44.275,158.260
C00672=1029.936,58.250,-96.341,168.380,44.273,158.260
C00673=1029.943,58.498,-96.358,168.382,44.271,158.260
C00674=1029.950,58.748,-96.375,168.385,44.269,158.260
C00675=1029.955,58.997,-96.392,168.387,44.267,158.259
C00676=1029.962,59.247,-96.410,168.390,44.265,158.259
C00677=1029.968,59.496,-96.427,168.392,44.264,158.259
C00678=1029.975,59.781,-96.447,168.395,44.261,158.259
C00679=1029.983,60.067,-96.466,168.398,44.259,158.259
C00680=1029.990,60.353,-96.486,168.400,44.257,158.259
C00681=1029.998,60.638,-96.506,168.403,44.254,158.258
C00682=1030.003,60.888,-96.523,168.405,44.253,158.258
C00683=1030.010,61.137,-96.540,168.408,44.251,158.258
C00684=1030.016,61.386,-96.557,168.410,44.249,158.258
C00685=1030.022,61.636,-96.575,168.413,44.247,158.258
C00686=1030.029,61.885,-96.592,168.415,44.245,158.258
C00687=1030.035,62.134,-96.609,168.417,44.243,158.258
C00688=1030.041,62.383,-96.627,168.420,44.241,158.257
C00689=1030.047,62.633,-96.644,168.422,44.239,158.257
C00690=1030.054,62.882,-96.661,168.425,44.237,158.257
C00691=1030.061,63.132,-96.678,168.427,44.235,158.257
C00692=1030.066,63.381,-96.696,168.429,44.233,158.257
C00693=1030.073,63.630,-96.713,168.431,44.231,158.257
C00694=1030.079,63.879,-96.731,168.434,44.229,158.256
C00695=1030.086,64.129,-96.748,168.437,44.227,158.256
C00696=1030.092,64.378,-96.766,168.438,44.226,158.256
C00697=1030.097,64.627,-96.784,168.441,44.224,158.256
C00698=1030.104,64.877,-96.801,168.443,44.222,158.256
C00699=1030.110,65.126,-96.818,168.446,44.220,158.256
C00700=1030.117,65.375,-96.836,168.448,44.218,158.256
C00701=1030.123,65.625,-96.854,168.450,44.216,158.255
C00702=1030.129,65.874,-96.871,168.453,44.214,158.255
C00703=1030.135,66.124,-96.889,168.455,44.212,158.255
C00704=1030.141,66.373,-96.906,168.458,44.210,158.255
C00705=1030.148,66.621,-96.924,168.460,44.209,158.255
C00706=1030.154,66.871,-96.942,168.462,44.207,158.255
C00707=1030.159,67.120,-96.960,168.465,44.205,158.255
C00708=1030.166,67.370,-96.977,168.467,44.203,158.254
C00709=1030.172,67.619,-96.995,168.469,44.202,158.254
C00710=1030.179,67.868,-97.012,168.472,44.200,158.254
C00711=1030.185,68.118,-97.030,168.474,44.198,158.254
C00712=1030.190,68.367,-97.047,168.477,44.196,158.254
C00713=1030.197,68.616,-97.066,168.479,44.194,158.254
C00714=1030.204,68.865,-97.083,168.481,44.193,158.254
C00715=1030.209,69.114,-97.101,168.484,44.191,158.254
C00716=1030.215,69.364,-97.119,168.486,44.189,158.253
C00717=1030.222,69.614,-97.136,168.488,44.187,158.253
C00718=1030.228,69.863,-97.154,168.490,44.185,158.253
C00719=1030.234,70.112,-97.173,168.493,44.183,158.253
C00720=1030.240,70.362,-97.190,168.496,44.181,158.253
C00721=1030.246,70.610,-97.207,168.497,44.180,158.253
C00722=1030.252,70.860,-97.225,168.500,44.178,158.253
C00723=1030.259,71.109,-97.244,168.502,44.176,158.252
C00724=1030.264,71.358,-97.262,168.505,44.174,158.252
C00725=1030.271,71.608,-97.279,168.507,44.173,158.252
C00726=1030.277,71.857,-97.297,168.509,44.171,158.252
C00727=1030.283,72.106,-97.315,168.512,44.169,158.252
C00728=1030.289,72.355,-97.333,168.515,44.167,158.252
C00729=1030.295,72.605,-97.351,168.516,44.165,158.252
C00730=1030.301,72.854,-97.369,168.519,44.163,158.252
C00731=1030.308,73.103,-97.387,168.521,44.161,158.251
C00732=1030.314,73.353,-97.405,168.524,44.160,158.251
C00733=1030.321,73.602,-97.423,168.526,44.158,158.251
C00734=1030.326,73.851,-97.441,168.528,44.156,158.251
C00735=1030.332,74.101,-97.459,168.531,44.154,158.251
C00736=1030.339,74.350,-97.477,168.533,44.152,158.251
C00737=1030.345,74.599,-97.494,168.535,44.150,158.251
C00738=1030.351,74.848,-97.512,168.538,44.148,158.250
C00739=1030.358,75.097,-97.531,168.540,44.147,158.250
C00740=1030.364,75.347,-97.549,168.543,44.145,158.250
C00741=1030.369,75.596,-97.567,168.545,44.143,158.250
C00742=1030.376,75.882,-97.587,168.548,44.141,158.250
C00743=1030.384,76.167,-97.608,168.551,44.139,158.250
C00744=1030.391,76.452,-97.628,168.553,44.137,158.250
C00745=1030.398,76.737,-97.649,168.556,44.134,158.249
C00746=1030.405,76.987,-97.668,168.558,44.133,158.249
C00747=1030.411,77.236,-97.686,168.561,44.131,158.249
C00748=1030.417,77.486,-97.704,168.563,44.130,158.249
C00749=1030.423,77.734,-97.722,168.565,44.128,158.249
C00750=1030.429,77.984,-97.740,168.568,44.126,158.249
C00751=1030.435,78.233,-97.758,168.570,44.124,158.249
C00752=1030.441,78.483,-97.776,168.572,44.122,158.248
C00753=1030.447,78.731,-97.795,168.574,44.120,158.248
C00754=1030.454,78.981,-97.813,168.577,44.118,158.248
C00755=1030.459,79.231,-97.832,168.580,44.117,158.248
C00756=1030.465,79.480,-97.850,168.581,44.115,158.248
C00757=1030.471,79.729,-97.868,168.584,44.113,158.248
C00758=1030.477,79.978,-97.887,168.587,44.112,158.248
C00759=1030.484,80.228,-97.905,168.589,44.110,158.248
C00760=1030.490,80.477,-97.923,168.591,44.108,158.247
C00761=1030.496,80.726,-97.942,168.593,44.106,158.247
C00762=1030.502,80.975,-97.959,168.596,44.105,158.247
C00763=1030.508,81.224,-97.978,168.598,44.103,158.247
C00764=1030.515,81.473,-97.997,168.600,44.101,158.247
C00765=1030.520,81.723,-98.015,168.603,44.099,158.247
C00766=1030.527,81.972,-98.034,168.606,44.097,158.247
C00767=1030.532,82.221,-98.052,168.607,44.096,158.246
C00768=1030.539,82.471,-98.070,168.610,44.094,158.246
C00769=1030.545,82.720,-98.089,168.612,44.092,158.246
C00770=1030.551,82.969,-98.107,168.615,44.091,158.246
C00771=1030.557,83.219,-98.125,168.617,44.089,158.246
C00772=1030.564,83.468,-98.144,168.619,44.087,158.246
C00773=1030.569,83.717,-98.162,168.622,44.085,158.246
C00774=1030.575,83.966,-98.181,168.625,44.083,158.246
C00775=1030.582,84.215,-98.200,168.626,44.081,158.245
C00776=1030.588,84.464,-98.218,168.629,44.080,158.245
C00777=1030.594,84.714,-98.236,168.631,44.078,158.245
C00778=1030.601,84.963,-98.255,168.634,44.076,158.245
C00779=1030.607,85.212,-98.273,168.637,44.074,158.245
C00780=1030.613,85.461,-98.292,168.638,44.072,158.245
C00781=1030.619,85.710,-98.310,168.641,44.071,158.245
C00782=1030.625,85.960,-98.329,168.644,44.069,158.245
C00783=1030.631,86.209,-98.347,168.646,44.067,158.244
C00784=1030.637,86.458,-98.366,168.648,44.065,158.244
C00785=1030.644,86.708,-98.384,168.650,44.063,158.244
C00786=1030.650,86.957,-98.403,168.653,44.062,158.244
C00787=1030.656,87.206,-98.421,168.656,44.060,158.244
C00788=1030.663,87.455,-98.440,168.657,44.058,158.244
C00789=1030.668,87.705,-98.459,168.660,44.056,158.244
C00790=1030.675,87.954,-98.477,168.662,44.054,158.243
C00791=1030.680,88.203,-98.495,168.665,44.052,158.243
C00792=1030.687,88.452,-98.514,168.668,44.050,158.243
C00793=1030.693,88.701,-98.533,168.669,44.049,158.243
C00794=1030.700,88.950,-98.551,168.672,44.047,158.243
C00795=1030.706,89.200,-98.569,168.674,44.045,158.243
C00796=1030.712,89.449,-98.588,168.677,44.043,158.243
C00797=1030.718,89.699,-98.607,168.680,44.041,158.242
C00798=1030.724,89.948,-98.626,168.681,44.040,158.242
C00799=1030.731,90.197,-98.645,168.684,44.038,158.242
C00800=1030.737,90.446,-98.664,168.687,44.036,158.242
C00801=1030.743,90.695,-98.682,168.688,44.034,158.242
C00802=1030.749,90.945,-98.702,168.691,44.033,158.242
C00803=1030.755,91.194,-98.720,168.694,44.031,158.242
C00804=1030.761,91.443,-98.740,168.696,44.029,158.242
C00805=1030.767,91.692,-98.758,168.698,44.028,158.241
C00806=1030.774,91.978,-98.779,168.701,44.026,158.241
C00807=1030.781,92.263,-98.801,168.704,44.024,158.241
C00808=1030.788,92.548,-98.823,168.707,44.022,158.241
C00809=1030.795,92.833,-98.844,168.709,44.020,158.241
C00810=1030.800,93.083,-98.863,168.712,44.018,158.241
C00811=1030.807,93.332,-98.882,168.713,44.016,158.241
C00812=1030.812,93.581,-98.901,168.716,44.014,158.240
C00813=1030.819,93.830,-98.920,168.719,44.013,158.240
C00814=1030.825,94.080,-98.939,168.721,44.011,158.240
C00815=1030.831,94.328,-98.958,168.724,44.009,158.240
C00816=1030.838,94.578,-98.977,168.726,44.008,158.240
C00817=1030.843,94.827,-98.996,168.728,44.006,158.240
C00818=1030.850,95.076,-99.015,168.731,44.004,158.240
C00819=1030.856,95.326,-99.034,168.733,44.002,158.240
C00820=1030.862,95.575,-99.053,168.735,44.000,158.239
C00821=1030.868,95.824,-99.072,168.738,43.998,158.239
C00822=1030.874,96.073,-99.091,168.740,43.996,158.239
C00823=1030.880,96.322,-99.109,168.743,43.995,158.239
C00824=1030.886,96.572,-99.129,168.745,43.994,158.239
C00825=1030.893,96.820,-99.148,168.747,43.992,158.239
C00826=1030.899,97.070,-99.167,168.750,43.990,158.239
C00827=1030.905,97.319,-99.186,168.752,43.988,158.239
C00828=1030.911,97.568,-99.205,168.755,43.986,158.238
C00829=1030.917,97.817,-99.224,168.757,43.984,158.238
C00830=1030.923,98.067,-99.243,168.759,43.982,158.238
C00831=1030.930,98.316,-99.263,168.762,43.981,158.238
C00832=1030.937,98.565,-99.281,168.765,43.979,158.238
C00833=1030.942,98.815,-99.301,168.767,43.977,158.238
C00834=1030.949,99.064,-99.319,168.769,43.976,158.238
C00835=1030.954,99.313,-99.339,168.771,43.974,158.237
C00836=1030.961,99.562,-99.358,168.774,43.972,158.237
C00837=1030.967,99.811,-99.377,168.777,43.970,158.237
C00838=1030.973,100.060,-99.396,168.778,43.968,158.237
C00839=1030.979,100.310,-99.415,168.781,43.967,158.237
C00840=1030.985,100.558,-99.435,168.784,43.965,158.237
C00841=1030.991,100.808,-99.454,168.786,43.963,158.237
C00842=1030.998,101.058,-99.473,168.788,43.962,158.237
C00843=1031.004,101.306,-99.493,168.791,43.960,158.237
C00844=1031.009,101.556,-99.513,168.793,43.958,158.236
C00845=1031.016,101.805,-99.531,168.796,43.957,158.236
C00846=1031.022,102.054,-99.551,168.797,43.955,158.236
C00847=1031.027,102.303,-99.570,168.800,43.954,158.236
C00848=1031.033,102.552,-99.590,168.803,43.952,158.236
C00849=1031.040,102.801,-99.609,168.805,43.950,158.236
C00850=1031.046,103.051,-99.628,168.808,43.948,158.236
C00851=1031.052,103.299,-99.648,168.810,43.946,158.236
C00852=1031.057,103.549,-99.667,168.812,43.945,158.236
C00853=1031.064,103.797,-99.687,168.815,43.943,158.235
C00854=1031.070,104.048,-99.706,168.818,43.941,158.235
C00855=1031.076,104.297,-99.726,168.819,43.940,158.235
C00856=1031.082,104.546,-99.746,168.822,43.938,158.235
C00857=1031.088,104.795,-99.764,168.825,43.936,158.235
C00858=1031.094,105.044,-99.784,168.827,43.935,158.235
C00859=1031.100,105.293,-99.803,168.830,43.933,158.235
C00860=1031.106,105.542,-99.823,168.831,43.931,158.234
C00861=1031.113,105.792,-99.842,168.834,43.930,158.234
C00862=1031.119,106.041,-99.862,168.837,43.928,158.234
C00863=1031.125,106.290,-99.882,168.839,43.926,158.234
C00864=1031.131,106.539,-99.902,168.841,43.924,158.234
C00865=1031.137,106.788,-99.920,168.844,43.922,158.234
C00866=1031.143,107.037,-99.940,168.846,43.921,158.234
C00867=1031.149,107.287,-99.960,168.849,43.919,158.234
C00868=1031.155,107.536,-99.980,168.852,43.917,158.234
C00869=1031.162,107.785,-99.998,168.853,43.916,158.233
C00870=1031.169,108.070,-100.020,168.857,43.914,158.233
C00871=1031.176,108.355,-100.044,168.859,43.912,158.233
C00872=1031.183,108.640,-100.066,168.862,43.910,158.233
C00873=1031.190,108.926,-100.088,168.865,43.908,158.233
C00874=1031.196,109.175,-100.108,168.867,43.906,158.233
C00875=1031.202,109.424,-100.128,168.870,43.904,158.233
C00876=1031.209,109.673,-100.147,168.872,43.902,158.232
C00877=1031.215,109.923,-100.167,168.875,43.900,158.232
C00878=1031.221,110.172,-100.187,168.877,43.899,158.232
C00879=1031.227,110.420,-100.206,168.879,43.897,158.232
C00880=1031.233,110.671,-100.226,168.882,43.896,158.232
C00881=1031.239,110.919,-100.246,168.885,43.894,158.232
C00882=1031.245,111.168,-100.266,168.887,43.892,158.232
C00883=1031.251,111.418,-100.285,168.889,43.891,158.232
C00884=1031.257,111.666,-100.305,168.892,43.889,158.231
C00885=1031.264,111.916,-100.325,168.894,43.887,158.231
C00886=1031.270,112.165,-100.344,168.897,43.885,158.231
C00887=1031.276,112.414,-100.364,168.900,43.884,158.231
C00888=1031.282,112.663,-100.384,168.901,43.882,158.231
C00889=1031.288,112.913,-100.404,168.904,43.880,158.231
C00890=1031.294,113.162,-100.424,168.907,43.879,158.231
C00891=1031.300,113.410,-100.444,168.909,43.877,158.231
C00892=1031.305,113.660,-100.464,168.912,43.875,158.231
C00893=1031.312,113.909,-100.485,168.914,43.874,158.231
C00894=1031.318,114.158,-100.504,168.916,43.872,158.230
C00895=1031.323,114.407,-100.524,168.919,43.870,158.230
C00896=1031.329,114.656,-100.544,168.922,43.869,158.230
C00897=1031.335,114.906,-100.565,168.923,43.868,158.230
C00898=1031.341,115.155,-100.585,168.926,43.866,158.230
C00899=1031.347,115.404,-100.605,168.929,43.864,158.230
C00900=1031.353,115.652,-100.624,168.931,43.863,158.230
C00901=1031.359,115.902,-100.645,168.933,43.862,158.230
C00902=1031.365,116.151,-100.665,168.936,43.860,158.230
C00903=1031.371,116.400,-100.685,168.938,43.858,158.229
C00904=1031.377,116.649,-100.705,168.941,43.857,158.229
C00905=1031.383,116.899,-100.725,168.944,43.855,158.229
C00906=1031.389,117.148,-100.745,168.945,43.853,158.229
C00907=1031.395,117.397,-100.765,168.948,43.852,158.229
C00908=1031.401,117.646,-100.785,168.951,43.850,158.229
C00909=1031.407,117.895,-100.806,168.954,43.849,158.229
C00910=1031.413,118.144,-100.826,168.956,43.847,158.229
C00911=1031.418,118.393,-100.846,168.958,43.845,158.229
C00912=1031.425,118.643,-100.867,168.961,43.844,158.229
C00913=1031.431,118.891,-100.886,168.963,43.842,158.229
C00914=1031.437,119.140,-100.906,168.966,43.840,158.228
C00915=1031.443,119.390,-100.927,168.969,43.839,158.228
C00916=1031.449,119.639,-100.947,168.970,43.837,158.228
C00917=1031.455,119.888,-100.967,168.973,43.835,158.228
C00918=1031.462,120.137,-100.988,168.976,43.834,158.228
C00919=1031.468,120.386,-101.008,168.978,43.832,158.228
C00920=1031.473,120.635,-101.028,168.981,43.830,158.228
C00921=1031.479,120.885,-101.048,168.984,43.829,158.228
C00922=1031.485,121.133,-101.068,168.985,43.827,158.228
C00923=1031.491,121.382,-101.088,168.988,43.826,158.227
C00924=1031.497,121.632,-101.109,168.991,43.824,158.227
C00925=1031.503,121.880,-101.130,168.993,43.822,158.227
C00926=1031.510,122.130,-101.150,168.996,43.821,158.227
C00927=1031.516,122.379,-101.170,168.999,43.819,158.227
C00928=1031.521,122.628,-101.191,169.000,43.818,158.227
C00929=1031.528,122.877,-101.211,169.003,43.816,158.227
C00930=1031.534,123.126,-101.231,169.006,43.814,158.227
C00931=1031.541,123.376,-101.251,169.008,43.813,158.227
C00932=1031.546,123.625,-101.272,169.011,43.811,158.226
C00933=1031.552,123.873,-101.292,169.014,43.809,158.226
C00934=1031.559,124.159,-101.316,169.016,43.807,158.226
C00935=1031.567,124.444,-101.339,169.019,43.805,158.226
C00936=1031.573,124.729,-101.362,169.022,43.804,158.226
C00937=1031.580,125.014,-101.386,169.025,43.802,158.226
C00938=1031.587,125.264,-101.406,169.028,43.800,158.226
C00939=1031.593,125.512,-101.426,169.029,43.798,158.226
C00940=1031.598,125.761,-101.447,169.032,43.796,158.225
C00941=1031.605,126.010,-101.467,169.035,43.795,158.225
C00942=1031.611,126.259,-101.487,169.037,43.793,158.225
C00943=1031.617,126.509,-101.508,169.040,43.791,158.225
C00944=1031.623,126.758,-101.528,169.043,43.790,158.225
C00945=1031.629,127.007,-101.549,169.045,43.788,158.225
C00946=1031.635,127.255,-101.569,169.048,43.787,158.225
C00947=1031.642,127.505,-101.590,169.051,43.785,158.225
C00948=1031.647,127.754,-101.610,169.053,43.784,158.225
C00949=1031.654,128.003,-101.631,169.055,43.782,158.225
C00950=1031.660,128.252,-101.651,169.058,43.780,158.224
C00951=1031.667,128.501,-101.671,169.061,43.779,158.224
C00952=1031.672,128.750,-101.693,169.063,43.777,158.224
C00953=1031.679,128.999,-101.713,169.066,43.775,158.224
C00954=1031.685,129.248,-101.733,169.068,43.773,158.224
C00955=1031.692,129.498,-101.753,169.071,43.772,158.224
C00956=1031.697,129.746,-101.775,169.074,43.770,158.224
C00957=1031.704,129.996,-101.795,169.076,43.768,158.224
C00958=1031.710,130.245,-101.815,169.079,43.767,158.224
C00959=1031.716,130.494,-101.837,169.081,43.765,158.223
C00960=1031.722,130.743,-101.857,169.083,43.763,158.223
C00961=1031.728,130.992,-101.878,169.086,43.762,158.223
C00962=1031.735,131.241,-101.898,169.089,43.760,158.223
C00963=1031.740,131.490,-101.919,169.092,43.759,158.223
C00964=1031.747,131.739,-101.940,169.094,43.757,158.223
C00965=1031.752,131.988,-101.961,169.097,43.755,158.223
C00966=1031.758,132.238,-101.982,169.100,43.754,158.223
C00967=1031.764,132.486,-102.002,169.101,43.752,158.223
C00968=1031.770,132.736,-102.024,169.104,43.751,158.223
C00969=1031.776,132.984,-102.044,169.107,43.749,158.223
C00970=1031.782,133.234,-102.065,169.110,43.748,158.223
C00971=1031.788,133.483,-102.086,169.112,43.746,158.222
C00972=1031.795,133.732,-102.107,169.115,43.745,158.222
C00973=1031.800,133.980,-102.128,169.118,43.743,158.222
C00974=1031.807,134.230,-102.149,169.120,43.741,158.222
C00975=1031.812,134.478,-102.170,169.122,43.740,158.222
C00976=1031.818,134.728,-102.191,169.125,43.738,158.222
C00977=1031.825,134.977,-102.212,169.127,43.737,158.222
C00978=1031.830,135.226,-102.232,169.130,43.735,158.222
C00979=1031.837,135.475,-102.253,169.133,43.734,158.222
C00980=1031.843,135.723,-102.275,169.135,43.732,158.222
C00981=1031.849,135.973,-102.296,169.138,43.730,158.221
C00982=1031.856,136.222,-102.317,169.141,43.729,158.221
C00983=1031.861,136.471,-102.337,169.143,43.727,158.221
C00984=1031.867,136.720,-102.359,169.146,43.726,158.221
C00985=1031.873,136.969,-102.380,169.149,43.724,158.221
C00986=1031.879,137.219,-102.400,169.151,43.723,158.221
C00987=1031.885,137.468,-102.422,169.153,43.721,158.221
C00988=1031.892,137.716,-102.443,169.156,43.720,158.221
C00989=1031.897,137.966,-102.464,169.159,43.718,158.221
C00990=1031.903,138.214,-102.485,169.161,43.716,158.221
C00991=1031.910,138.463,-102.506,169.164,43.715,158.221
C00992=1031.916,138.713,-102.527,169.167,43.713,158.221
C00993=1031.921,138.961,-102.548,169.170,43.712,158.221
C00994=1031.928,139.211,-102.570,169.172,43.710,158.220
C00995=1031.934,139.460,-102.591,169.175,43.709,158.220
C00996=1031.940,139.708,-102.612,169.178,43.707,158.220
C00997=1031.946,139.958,-102.633,169.179,43.706,158.220
C00998=1031.952,140.243,-102.658,169.183,43.704,158.220
C00999=1031.960,140.528,-102.682,169.186,43.703,158.220
C01000=1031.967,140.813,-102.706,169.189,43.701,158.220
C01001=1031.973,141.097,-102.731,169.192,43.699,158.220
C01002=1031.979,141.347,-102.752,169.195,43.698,158.220
C01003=1031.985,141.596,-102.774,169.198,43.696,158.220
C01004=1031.991,141.844,-102.795,169.200,43.695,158.220
C01005=1031.998,142.093,-102.816,169.203,43.693,158.220
C01006=1032.004,142.343,-102.838,169.205,43.692,158.219
C01007=1032.009,142.592,-102.858,169.208,43.691,158.219
C01008=1032.015,142.841,-102.880,169.210,43.689,158.219
C01009=1032.021,143.090,-102.902,169.213,43.687,158.219
C01010=1032.027,143.339,-102.923,169.216,43.686,158.219
C01011=1032.034,143.587,-102.944,169.219,43.684,158.219
C01012=1032.040,143.837,-102.966,169.221,43.683,158.219
C01013=1032.046,144.086,-102.987,169.224,43.681,158.219
C01014=1032.052,144.334,-103.009,169.227,43.679,158.219
C01015=1032.058,144.584,-103.030,169.229,43.678,158.219
C01016=1032.064,144.833,-103.052,169.232,43.676,158.219
C01017=1032.070,145.082,-103.073,169.235,43.675,158.219
C01018=1032.076,145.330,-103.095,169.237,43.673,158.219
C01019=1032.082,145.580,-103.116,169.240,43.672,158.219
C01020=1032.089,145.829,-103.137,169.243,43.670,158.218
C01021=1032.095,146.078,-103.159,169.246,43.669,158.218
C01022=1032.100,146.326,-103.180,169.248,43.667,158.218
C01023=1032.107,146.575,-103.202,169.251,43.666,158.218
C01024=1032.113,146.825,-103.224,169.254,43.665,158.218
C01025=1032.119,147.074,-103.245,169.257,43.663,158.218
C01026=1032.124,147.322,-103.266,169.259,43.662,158.218
C01027=1032.131,147.572,-103.288,169.262,43.660,158.218
C01028=1032.137,147.821,-103.310,169.265,43.659,158.218
C01029=1032.143,148.070,-103.331,169.268,43.657,158.218
C01030=1032.149,148.319,-103.353,169.269,43.656,158.218
C01031=1032.154,148.568,-103.375,169.272,43.655,158.218
C01032=1032.160,148.817,-103.397,169.275,43.653,158.218
C01033=1032.167,149.066,-103.419,169.277,43.651,158.218
C01034=1032.173,149.315,-103.440,169.280,43.650,158.218
C01035=1032.178,149.564,-103.462,169.283,43.648,158.217
C01036=1032.184,149.813,-103.483,169.286,43.647,158.217
C01037=1032.191,150.061,-103.506,169.289,43.646,158.217
C01038=1032.197,150.311,-103.527,169.291,43.644,158.217
C01039=1032.202,150.559,-103.549,169.294,43.643,158.217
C01040=1032.208,150.809,-103.571,169.297,43.642,158.217
C01041=1032.214,151.058,-103.593,169.299,43.640,158.217
C01042=1032.221,151.306,-103.615,169.302,43.639,158.217
C01043=1032.227,151.556,-103.637,169.305,43.637,158.217
C01044=1032.233,151.805,-103.658,169.308,43.636,158.217
C01045=1032.239,152.053,-103.679,169.310,43.634,158.217
C01046=1032.244,152.302,-103.702,169.313,43.633,158.217
C01047=1032.251,152.551,-103.724,169.316,43.631,158.217
C01048=1032.257,152.801,-103.746,169.319,43.630,158.217
C01049=1032.263,153.049,-103.768,169.322,43.629,158.217
C01050=1032.269,153.298,-103.790,169.324,43.627,158.217
C01051=1032.275,153.548,-103.811,169.327,43.626,158.217
C01052=1032.281,153.796,-103.834,169.330,43.625,158.217
C01053=1032.287,154.045,-103.855,169.332,43.623,158.216
C01054=1032.293,154.294,-103.877,169.335,43.622,158.216
C01055=1032.299,154.543,-103.899,169.338,43.620,158.216
C01056=1032.305,154.792,-103.922,169.341,43.619,158.216
C01057=1032.311,155.041,-103.944,169.344,43.617,158.216
C01058=1032.317,155.290,-103.966,169.346,43.616,158.216
C01059=1032.322,155.539,-103.988,169.349,43.615,158.216
C01060=1032.329,155.787,-104.010,169.352,43.613,158.216
C01061=1032.335,156.037,-104.032,169.355,43.612,158.216
C01062=1032.342,156.321,-104.057,169.358,43.610,158.216
C01063=1032.348,156.606,-104.082,169.361,43.609,158.216
C01064=1032.355,156.891,-104.108,169.365,43.607,158.216
C01065=1032.363,157.175,-104.133,169.367,43.605,158.216
C01066=1032.368,157.424,-104.155,169.370,43.604,158.216
C01067=1032.375,157.673,-104.178,169.373,43.603,158.216
C01068=1032.381,157.922,-104.199,169.376,43.601,158.216
C01069=1032.387,158.171,-104.222,169.379,43.600,158.216
C01070=1032.393,158.420,-104.244,169.381,43.599,158.216
C01071=1032.399,158.669,-104.266,169.385,43.597,158.216
C01072=1032.405,158.918,-104.288,169.388,43.595,158.216
C01073=1032.411,159.167,-104.311,169.391,43.594,158.216
C01074=1032.417,159.416,-104.332,169.393,43.593,158.216
C01075=1032.423,159.665,-104.355,169.396,43.592,158.216
C01076=1032.430,159.914,-104.378,169.399,43.590,158.215
C01077=1032.435,160.163,-104.400,169.402,43.589,158.215
C01078=1032.441,160.412,-104.423,169.405,43.588,158.215
C01079=1032.446,160.661,-104.446,169.407,43.586,158.215
C01080=1032.453,160.910,-104.467,169.410,43.585,158.215
C01081=1032.458,161.158,-104.490,169.413,43.584,158.215
C01082=1032.463,161.407,-104.513,169.416,43.583,158.215
C01083=1032.470,161.656,-104.535,169.419,43.582,158.215
C01084=1032.476,161.905,-104.558,169.422,43.580,158.215
C01085=1032.481,162.154,-104.580,169.424,43.579,158.215
C01086=1032.487,162.403,-104.603,169.427,43.578,158.215
C01087=1032.493,162.652,-104.626,169.430,43.577,158.215
C01088=1032.499,162.901,-104.649,169.433,43.576,158.215
C01089=1032.505,163.149,-104.672,169.436,43.574,158.215
C01090=1032.510,163.399,-104.694,169.438,43.573,158.215
C01091=1032.517,163.648,-104.716,169.441,43.572,158.215
C01092=1032.522,163.896,-104.739,169.444,43.571,158.215
C01093=1032.528,164.145,-104.762,169.447,43.570,158.215
C01094=1032.534,164.394,-104.785,169.450,43.568,158.215
C01095=1032.540,164.643,-104.807,169.453,43.567,158.215
C01096=1032.546,164.892,-104.830,169.455,43.566,158.215
C01097=1032.552,165.141,-104.853,169.458,43.565,158.215
C01098=1032.557,165.390,-104.875,169.461,43.564,158.215
C01099=1032.563,165.639,-104.898,169.464,43.562,158.215
C01100=1032.569,165.888,-104.921,169.467,43.561,158.215
C01101=1032.575,166.137,-104.944,169.471,43.560,158.215
C01102=1032.581,166.385,-104.967,169.473,43.559,158.215
C01103=1032.587,166.634,-104.990,169.476,43.557,158.215
C01104=1032.593,166.883,-105.012,169.479,43.556,158.215
C01105=1032.599,167.132,-105.035,169.482,43.554,158.215
C01106=1032.605,167.381,-105.058,169.484,43.553,158.215
C01107=1032.610,167.630,-105.081,169.487,43.552,158.215
C01108=1032.617,167.878,-105.103,169.490,43.551,158.215
C01109=1032.623,168.128,-105.126,169.493,43.550,158.215
C01110=1032.629,168.377,-105.149,169.496,43.548,158.215
C01111=1032.635,168.626,-105.172,169.499,43.547,158.215
C01112=1032.640,168.874,-105.195,169.502,43.546,158.215
C01113=1032.647,169.123,-105.218,169.505,43.545,158.215
C01114=1032.652,169.372,-105.241,169.508,43.543,158.215
C01115=1032.658,169.621,-105.264,169.511,43.542,158.215
C01116=1032.664,169.870,-105.286,169.514,43.541,158.215
C01117=1032.670,170.118,-105.309,169.517,43.540,158.215
C01118=1032.677,170.368,-105.332,169.519,43.539,158.215
C01119=1032.683,170.616,-105.356,169.522,43.537,158.215
C01120=1032.688,170.865,-105.379,169.525,43.536,158.215
C01121=1032.694,171.114,-105.402,169.529,43.535,158.215
C01122=1032.701,171.363,-105.424,169.532,43.534,158.215
C01123=1032.706,171.611,-105.447,169.535,43.532,158.215
C01124=1032.712,171.860,-105.470,169.537,43.531,158.215
C01125=1032.718,172.110,-105.493,169.540,43.530,158.215
C01126=1032.726,172.394,-105.520,169.544,43.529,158.215
C01127=1032.733,172.678,-105.545,169.547,43.528,158.215
C01128=1032.739,172.962,-105.572,169.551,43.526,158.215
C01129=1032.746,173.246,-105.599,169.555,43.525,158.215
C01130=1032.752,173.495,-105.622,169.557,43.524,158.215
C01131=1032.758,173.744,-105.645,169.560,43.522,158.215
C01132=1032.765,173.993,-105.667,169.563,43.521,158.215
C01133=1032.771,174.242,-105.691,169.566,43.520,158.215
C01134=1032.776,174.490,-105.714,169.570,43.519,158.215
C01135=1032.782,174.739,-105.737,169.572,43.517,158.215
C01136=1032.789,174.989,-105.760,169.575,43.516,158.215
C01137=1032.795,175.237,-105.783,169.578,43.515,158.215
C01138=1032.801,175.486,-105.806,169.581,43.514,158.215
C01139=1032.807,175.735,-105.829,169.585,43.512,158.215
C01140=1032.813,175.984,-105.852,169.588,43.511,158.215
C01141=1032.819,176.233,-105.876,169.590,43.510,158.215
C01142=1032.825,176.482,-105.899,169.593,43.509,158.215
C01143=1032.832,176.731,-105.922,169.596,43.508,158.215
C01144=1032.838,176.979,-105.945,169.600,43.506,158.215
C01145=1032.844,177.228,-105.968,169.603,43.505,158.215
C01146=1032.849,177.477,-105.991,169.606,43.504,158.215
C01147=1032.856,177.726,-106.015,169.608,43.503,158.215
C01148=1032.862,177.975,-106.038,169.612,43.501,158.215
C01149=1032.868,178.223,-106.061,169.615,43.500,158.215
C01150=1032.875,178.472,-106.085,169.618,43.499,158.215
C01151=1032.881,178.721,-106.108,169.621,43.498,158.215
C01152=1032.887,178.969,-106.131,169.625,43.496,158.215
C01153=1032.893,179.219,-106.155,169.627,43.495,158.215
C01154=1032.899,179.468,-106.178,169.630,43.494,158.215
C01155=1032.906,179.716,-106.201,169.633,43.493,158.215
C01156=1032.912,179.966,-106.224,169.637,43.491,158.215
C01157=1032.918,180.214,-106.248,169.640,43.490,158.215
C01158=1032.924,180.463,-106.271,169.643,43.489,158.215
C01159=1032.930,180.712,-106.295,169.645,43.488,158.215
C01160=1032.936,180.961,-106.318,169.649,43.487,158.215
C01161=1032.943,181.209,-106.341,169.652,43.486,158.215
C01162=1032.949,181.458,-106.364,169.655,43.485,158.215
C01163=1032.956,181.707,-106.388,169.659,43.483,158.215
C01164=1032.961,181.956,-106.411,169.662,43.482,158.215
C01165=1032.968,182.204,-106.435,169.665,43.481,158.215
C01166=1032.974,182.454,-106.458,169.667,43.480,158.215
C01167=1032.980,182.702,-106.482,169.671,43.478,158.215
C01168=1032.987,182.951,-106.504,169.674,43.477,158.215
C01169=1032.992,183.200,-106.528,169.677,43.476,158.215
C01170=1032.999,183.449,-106.553,169.680,43.476,158.215
C01171=1033.005,183.697,-106.576,169.684,43.474,158.215
C01172=1033.010,183.947,-106.600,169.687,43.473,158.215
C01173=1033.017,184.196,-106.624,169.690,43.472,158.216
C01174=1033.022,184.444,-106.648,169.692,43.471,158.216
C01175=1033.028,184.692,-106.672,169.696,43.470,158.216
C01176=1033.034,184.942,-106.696,169.699,43.469,158.216
C01177=1033.040,185.191,-106.719,169.702,43.468,158.216
C01178=1033.046,185.439,-106.743,169.705,43.468,158.216
C01179=1033.051,185.688,-106.768,169.709,43.466,158.216
C01180=1033.058,185.936,-106.791,169.712,43.466,158.216
C01181=1033.063,186.186,-106.816,169.715,43.464,158.216
C01182=1033.069,186.434,-106.839,169.718,43.463,158.216
C01183=1033.075,186.683,-106.864,169.722,43.463,158.216
C01184=1033.081,186.932,-106.888,169.725,43.461,158.216
C01185=1033.087,187.180,-106.912,169.728,43.461,158.216
C01186=1033.093,187.430,-106.935,169.730,43.460,158.216
C01187=1033.099,187.678,-106.959,169.734,43.458,158.216
C01188=1033.105,187.927,-106.984,169.737,43.458,158.216
C01189=1033.111,188.176,-107.007,169.740,43.456,158.216
C01190=1033.118,188.459,-107.035,169.744,43.456,158.217
C01191=1033.125,188.743,-107.063,169.748,43.454,158.217
C01192=1033.132,189.027,-107.090,169.751,43.453,158.217
C01193=1033.138,189.311,-107.118,169.755,43.452,158.217
C01194=1033.144,189.560,-107.142,169.758,43.451,158.217
C01195=1033.150,189.809,-107.166,169.762,43.451,158.217
C01196=1033.156,190.057,-107.190,169.765,43.449,158.217
C01197=1033.162,190.306,-107.214,169.767,43.448,158.217
C01198=1033.168,190.554,-107.238,169.772,43.447,158.217
C01199=1033.174,190.804,-107.263,169.774,43.446,158.217
C01200=1033.180,191.052,-107.286,169.777,43.446,158.217
C01201=1033.186,191.301,-107.311,169.781,43.444,158.217
C01202=1033.193,191.550,-107.335,169.784,43.444,158.217
C01203=1033.198,191.798,-107.360,169.787,43.443,158.217
C01204=1033.205,192.047,-107.384,169.791,43.442,158.218
C01205=1033.210,192.296,-107.408,169.794,43.441,158.218
C01206=1033.217,192.545,-107.432,169.797,43.440,158.218
C01207=1033.222,192.793,-107.456,169.801,43.439,158.218
C01208=1033.229,193.042,-107.480,169.804,43.438,158.218
C01209=1033.235,193.292,-107.505,169.807,43.437,158.218
C01210=1033.241,193.539,-107.529,169.811,43.436,158.218
C01211=1033.247,193.789,-107.554,169.814,43.435,158.218
C01212=1033.253,194.037,-107.578,169.817,43.435,158.218
C01213=1033.259,194.286,-107.602,169.820,43.433,158.218
C01214=1033.266,194.535,-107.626,169.823,43.433,158.218
C01215=1033.271,194.783,-107.651,169.827,43.431,158.218
C01216=1033.278,195.032,-107.675,169.830,43.431,158.218
C01217=1033.284,195.281,-107.700,169.833,43.430,158.218
C01218=1033.290,195.530,-107.724,169.837,43.429,158.219
C01219=1033.296,195.778,-107.749,169.840,43.428,158.219
C01220=1033.303,196.027,-107.773,169.844,43.427,158.219
C01221=1033.308,196.276,-107.797,169.847,43.426,158.219
C01222=1033.314,196.525,-107.821,169.850,43.425,158.219
C01223=1033.321,196.773,-107.847,169.854,43.424,158.219
C01224=1033.327,197.022,-107.870,169.857,43.423,158.219
C01225=1033.333,197.271,-107.895,169.861,43.422,158.219
C01226=1033.340,197.519,-107.920,169.864,43.421,158.219
C01227=1033.345,197.768,-107.944,169.868,43.420,158.219
C01228=1033.352,198.017,-107.968,169.871,43.420,158.219
C01229=1033.358,198.266,-107.993,169.873,43.418,158.219
C01230=1033.364,198.515,-108.017,169.878,43.418,158.220
C01231=1033.370,198.763,-108.042,169.881,43.417,158.220
C01232=1033.377,199.012,-108.066,169.884,43.416,158.220
C01233=1033.383,199.261,-108.091,169.887,43.415,158.220
C01234=1033.389,199.509,-108.116,169.891,43.414,158.220
C01235=1033.395,199.758,-108.140,169.894,43.413,158.220
C01236=1033.402,200.006,-108.165,169.898,43.412,158.220
C01237=1033.408,200.255,-108.189,169.901,43.411,158.220
C01238=1033.414,200.504,-108.215,169.904,43.411,158.220
C01239=1033.420,200.753,-108.239,169.908,43.409,158.220
C01240=1033.426,201.001,-108.264,169.911,43.409,158.220
C01241=1033.432,201.250,-108.288,169.915,43.408,158.221
C01242=1033.438,201.499,-108.314,169.918,43.408,158.221
C01243=1033.444,201.748,-108.339,169.922,43.406,158.221
C01244=1033.450,201.996,-108.363,169.925,43.406,158.221
C01245=1033.456,202.245,-108.389,169.929,43.405,158.221
C01246=1033.463,202.493,-108.413,169.932,43.404,158.221
C01247=1033.469,202.743,-108.438,169.935,43.404,158.221
C01248=1033.475,202.991,-108.463,169.939,43.403,158.221
C01249=1033.481,203.239,-108.488,169.942,43.402,158.222
C01250=1033.486,203.488,-108.513,169.946,43.401,158.222
C01251=1033.493,203.737,-108.538,169.949,43.401,158.222
C01252=1033.499,203.986,-108.564,169.953,43.400,158.222
C01253=1033.505,204.234,-108.589,169.956,43.399,158.222
C01254=1033.531,205.284,-108.694,170.290,43.503,158.271
C01255=1033.541,205.629,-108.730,170.293,43.503,158.271
C01256=1033.550,205.974,-108.767,170.296,43.503,158.271
C01257=1033.559,206.319,-108.804,170.299,43.503,158.271
C01258=1033.569,206.664,-108.841,170.304,43.503,158.272
C01259=1033.575,206.912,-108.867,170.306,43.503,158.272
C01260=1033.582,207.161,-108.893,170.308,43.503,158.272
C01261=1033.589,207.409,-108.919,170.311,43.503,158.272
C01262=1033.595,207.658,-108.946,170.313,43.503,158.273
C01263=1033.602,207.907,-108.973,170.316,43.504,158.273
C01264=1033.609,208.155,-108.999,170.319,43.503,158.273
C01265=1033.616,208.404,-109.025,170.321,43.503,158.273
C01266=1033.622,208.652,-109.052,170.323,43.504,158.274
C01267=1033.629,208.901,-109.078,170.326,43.503,158.274
C01268=1033.636,209.149,-109.105,170.329,43.503,158.274
C01269=1033.643,209.397,-109.131,170.331,43.504,158.274
C01270=1033.649,209.646,-109.158,170.334,43.504,158.274
C01271=1033.656,209.895,-109.185,170.336,43.503,158.274
C01272=1033.663,210.143,-109.211,170.338,43.504,158.275
C01273=1033.669,210.392,-109.238,170.342,43.504,158.275
C01274=1033.677,210.640,-109.265,170.344,43.504,158.275
C01275=1033.683,210.888,-109.291,170.346,43.504,158.275
C01276=1033.689,211.137,-109.318,170.349,43.504,158.276
C01277=1033.697,211.386,-109.345,170.351,43.504,158.276
C01278=1033.702,211.634,-109.371,170.354,43.504,158.276
C01279=1033.710,211.883,-109.398,170.357,43.504,158.276
C01280=1033.716,212.132,-109.425,170.359,43.504,158.276
C01281=1033.723,212.380,-109.451,170.362,43.504,158.277
C01282=1033.729,212.628,-109.479,170.364,43.504,158.277
C01283=1033.736,212.877,-109.506,170.367,43.505,158.277
C01284=1033.742,213.125,-109.532,170.370,43.505,158.278
C01285=1033.750,213.373,-109.559,170.372,43.504,158.278
C01286=1033.756,213.622,-109.586,170.374,43.505,158.278
C01287=1033.763,213.870,-109.612,170.377,43.505,158.278
C01288=1033.769,214.119,-109.640,170.380,43.505,158.278
C01289=1033.776,214.368,-109.667,170.383,43.505,158.279
C01290=1033.782,214.616,-109.693,170.385,43.505,158.279
C01291=1033.789,214.864,-109.720,170.387,43.505,158.279
C01292=1033.796,215.113,-109.747,170.390,43.505,158.279
C01293=1033.803,215.361,-109.774,170.393,43.505,158.279
C01294=1033.809,215.610,-109.801,170.396,43.505,158.280
C01295=1033.816,215.858,-109.828,170.398,43.506,158.280
C01296=1033.823,216.107,-109.855,170.400,43.505,158.280
C01297=1033.830,216.356,-109.882,170.403,43.505,158.280
C01298=1033.836,216.603,-109.909,170.406,43.506,158.281
C01299=1033.843,216.852,-109.935,170.409,43.506,158.281
C01300=1033.850,217.101,-109.963,170.411,43.506,158.281
C01301=1033.857,217.349,-109.990,170.413,43.506,158.281
C01302=1033.863,217.597,-110.017,170.416,43.506,158.282
C01303=1033.870,217.846,-110.043,170.419,43.506,158.282
C01304=1033.877,218.094,-110.071,170.422,43.506,158.282
C01305=1033.884,218.343,-110.098,170.424,43.506,158.282
C01306=1033.891,218.591,-110.125,170.428,43.506,158.283
C01307=1033.897,218.840,-110.151,170.430,43.507,158.283
C01308=1033.904,219.088,-110.179,170.433,43.506,158.283
C01309=1033.911,219.337,-110.205,170.435,43.506,158.283
C01310=1033.918,219.585,-110.233,170.438,43.506,158.283
C01311=1033.926,219.936,-110.271,170.442,43.506,158.284
C01312=1033.936,220.287,-110.311,170.445,43.507,158.284
C01313=1033.946,220.637,-110.349,170.449,43.507,158.284
C01314=1033.955,220.988,-110.387,170.453,43.507,158.285
C01315=1033.961,221.236,-110.415,170.456,43.507,158.285
C01316=1033.968,221.485,-110.442,170.458,43.507,158.285
C01317=1033.974,221.734,-110.469,170.461,43.507,158.286
C01318=1033.982,221.982,-110.496,170.464,43.508,158.286
C01319=1033.988,222.231,-110.524,170.466,43.508,158.286
C01320=1033.995,222.478,-110.552,170.469,43.508,158.286
C01321=1034.001,222.727,-110.579,170.471,43.508,158.287
C01322=1034.008,222.976,-110.606,170.475,43.508,158.287
C01323=1034.015,223.224,-110.633,170.477,43.509,158.287
C01324=1034.022,223.472,-110.661,170.480,43.509,158.287
C01325=1034.028,223.721,-110.688,170.482,43.509,158.288
C01326=1034.035,223.970,-110.716,170.486,43.509,158.288
C01327=1034.041,224.218,-110.743,170.488,43.509,158.288
C01328=1034.048,224.466,-110.770,170.491,43.509,158.288
C01329=1034.055,224.714,-110.798,170.493,43.510,158.289
C01330=1034.061,224.963,-110.825,170.497,43.510,158.289
C01331=1034.068,225.212,-110.853,170.499,43.510,158.289
C01332=1034.075,225.460,-110.881,170.502,43.510,158.289
C01333=1034.082,225.708,-110.908,170.504,43.510,158.290
C01334=1034.089,225.957,-110.935,170.507,43.510,158.290
C01335=1034.095,226.205,-110.963,170.510,43.510,158.290
C01336=1034.102,226.454,-110.991,170.513,43.510,158.290
C01337=1034.109,226.702,-111.019,170.515,43.510,158.291
C01338=1034.115,226.951,-111.046,170.518,43.510,158.291
C01339=1034.123,227.199,-111.073,170.521,43.511,158.291
C01340=1034.129,227.447,-111.100,170.524,43.511,158.291
C01341=1034.135,227.695,-111.128,170.526,43.511,158.292
C01342=1034.142,227.944,-111.156,170.529,43.511,158.292
C01343=1034.149,228.192,-111.183,170.532,43.511,158.292
C01344=1034.155,228.441,-111.211,170.535,43.511,158.292
C01345=1034.162,228.689,-111.239,170.537,43.512,158.293
C01346=1034.169,228.938,-111.267,170.540,43.512,158.293
C01347=1034.175,229.186,-111.294,170.543,43.512,158.293
C01348=1034.182,229.434,-111.323,170.546,43.513,158.294
C01349=1034.189,229.682,-111.350,170.549,43.513,158.294
C01350=1034.196,229.931,-111.378,170.552,43.513,158.294
C01351=1034.202,230.179,-111.406,170.555,43.513,158.294
C01352=1034.209,230.428,-111.434,170.557,43.513,158.295
C01353=1034.216,230.676,-111.461,170.560,43.514,158.295
C01354=1034.223,230.924,-111.489,170.563,43.514,158.295
C01355=1034.228,231.173,-111.517,170.566,43.514,158.295
C01356=1034.235,231.422,-111.545,170.568,43.514,158.296
C01357=1034.242,231.670,-111.574,170.571,43.514,158.296
C01358=1034.249,231.918,-111.601,170.574,43.514,158.296
C01359=1034.255,232.166,-111.629,170.577,43.515,158.297
C01360=1034.262,232.415,-111.657,170.579,43.515,158.297
C01361=1034.268,232.663,-111.686,170.583,43.515,158.297
C01362=1034.275,232.911,-111.714,170.586,43.516,158.297
C01363=1034.282,233.160,-111.741,170.588,43.516,158.298
C01364=1034.288,233.408,-111.769,170.591,43.516,158.298
C01365=1034.295,233.656,-111.797,170.594,43.516,158.298
C01366=1034.301,233.905,-111.826,170.597,43.517,158.299
C01367=1034.311,234.248,-111.864,170.600,43.517,158.299
C01368=1034.320,234.591,-111.903,170.605,43.517,158.299
C01369=1034.329,234.934,-111.942,170.608,43.518,158.300
C01370=1034.339,235.277,-111.981,170.613,43.518,158.300
C01371=1034.345,235.526,-112.009,170.616,43.518,158.300
C01372=1034.352,235.774,-112.037,170.618,43.518,158.301
C01373=1034.359,236.023,-112.066,170.622,43.519,158.301
C01374=1034.365,236.272,-112.093,170.624,43.519,158.301
C01375=1034.372,236.519,-112.122,170.627,43.519,158.302
C01376=1034.378,236.768,-112.150,170.630,43.519,158.302
C01377=1034.385,237.016,-112.179,170.633,43.520,158.302
C01378=1034.392,237.264,-112.206,170.636,43.520,158.302
C01379=1034.399,237.513,-112.234,170.638,43.521,158.303
C01380=1034.405,237.761,-112.263,170.642,43.521,158.303
C01381=1034.412,238.009,-112.291,170.645,43.521,158.303
C01382=1034.419,238.258,-112.320,170.647,43.521,158.304
C01383=1034.426,238.506,-112.347,170.650,43.521,158.304
C01384=1034.432,238.755,-112.376,170.654,43.522,158.304
C01385=1034.439,239.003,-112.404,170.656,43.522,158.305
C01386=1034.446,239.251,-112.432,170.659,43.522,158.305
C01387=1034.452,239.500,-112.461,170.662,43.522,158.305
C01388=1034.459,239.748,-112.490,170.665,43.522,158.305
C01389=1034.466,239.996,-112.518,170.668,43.523,158.306
C01390=1034.472,240.245,-112.546,170.670,43.523,158.306
C01391=1034.479,240.492,-112.575,170.674,43.524,158.306
C01392=1034.486,240.741,-112.603,170.677,43.524,158.307
C01393=1034.492,240.989,-112.632,170.679,43.524,158.307
C01394=1034.499,241.237,-112.660,170.683,43.525,158.307
C01395=1034.506,241.486,-112.689,170.686,43.525,158.308
C01396=1034.513,241.734,-112.717,170.688,43.525,158.308
C01397=1034.519,241.982,-112.746,170.692,43.526,158.308
C01398=1034.525,242.230,-112.775,170.694,43.526,158.308
C01399=1034.532,242.479,-112.803,170.697,43.527,158.309
C01400=1034.539,242.728,-112.832,170.701,43.527,158.309
C01401=1034.546,242.975,-112.861,170.703,43.527,158.309
C01402=1034.552,243.224,-112.890,170.706,43.528,158.310
C01403=1034.559,243.472,-112.918,170.710,43.528,158.310
C01404=1034.565,243.720,-112.947,170.712,43.528,158.310
C01405=1034.573,243.969,-112.975,170.715,43.529,158.311
C01406=1034.579,244.217,-113.005,170.719,43.529,158.311
C01407=1034.586,244.465,-113.032,170.721,43.529,158.311
C01408=1034.592,244.713,-113.061,170.724,43.530,158.312
C01409=1034.598,244.962,-113.090,170.728,43.530,158.312
C01410=1034.605,245.210,-113.120,170.730,43.531,158.312
C01411=1034.612,245.458,-113.148,170.733,43.531,158.313
C01412=1034.618,245.706,-113.177,170.737,43.531,158.313
C01413=1034.624,245.954,-113.206,170.739,43.532,158.313
C01414=1034.631,246.203,-113.235,170.743,43.532,158.314
C01415=1034.637,246.451,-113.265,170.746,43.532,158.314
C01416=1034.644,246.699,-113.293,170.748,43.533,158.315
C01417=1034.651,246.947,-113.322,170.752,43.533,158.315
C01418=1034.657,247.196,-113.351,170.755,43.533,158.315
C01419=1034.664,247.444,-113.381,170.757,43.534,158.315
C01420=1034.670,247.692,-113.410,170.761,43.534,158.316
C01421=1034.676,247.941,-113.439,170.764,43.535,158.316
C01422=1034.683,248.188,-113.467,170.766,43.535,158.316
C01423=1034.692,248.526,-113.507,170.771,43.536,158.317
C01424=1034.701,248.863,-113.547,170.775,43.536,158.317
C01425=1034.710,249.201,-113.586,170.779,43.538,158.318
C01426=1034.719,249.538,-113.626,170.783,43.538,158.318
C01427=1034.726,249.786,-113.655,170.787,43.538,158.319
C01428=1034.732,250.035,-113.684,170.790,43.539,158.319
C01429=1034.738,250.283,-113.713,170.792,43.539,158.319
C01430=1034.746,250.531,-113.742,170.796,43.540,158.320
C01431=1034.752,250.779,-113.771,170.799,43.540,158.320
C01432=1034.759,251.028,-113.800,170.802,43.541,158.321
C01433=1034.766,251.276,-113.830,170.805,43.541,158.321
C01434=1034.772,251.524,-113.860,170.808,43.541,158.321
C01435=1034.778,251.772,-113.889,170.812,43.542,158.322
C01436=1034.786,252.021,-113.917,170.814,43.542,158.322
C01437=1034.792,252.268,-113.947,170.817,43.542,158.322
C01438=1034.799,252.517,-113.977,170.821,43.543,158.323
C01439=1034.805,252.765,-114.006,170.824,43.543,158.323
C01440=1034.812,253.013,-114.035,170.827,43.544,158.323
C01441=1034.819,253.261,-114.065,170.830,43.544,158.324
C01442=1034.825,253.509,-114.094,170.833,43.545,158.324
C01443=1034.833,253.758,-114.123,170.837,43.545,158.324
C01444=1034.839,254.006,-114.152,170.840,43.546,158.325
C01445=1034.846,254.254,-114.182,170.842,43.546,158.325
C01446=1034.852,254.502,-114.211,170.846,43.547,158.325
C01447=1034.859,254.751,-114.240,170.849,43.547,158.326
C01448=1034.866,254.999,-114.270,170.852,43.547,158.326
C01449=1034.872,255.247,-114.299,170.856,43.548,158.327
C01450=1034.880,255.495,-114.329,170.858,43.548,158.327
C01451=1034.886,255.743,-114.358,170.862,43.549,158.327
C01452=1034.893,255.992,-114.387,170.865,43.549,158.328
C01453=1034.900,256.239,-114.417,170.868,43.550,158.328
C01454=1034.906,256.488,-114.446,170.872,43.550,158.328
C01455=1034.913,256.736,-114.476,170.874,43.551,158.329
C01456=1034.920,256.985,-114.505,170.878,43.551,158.329
C01457=1034.927,257.232,-114.534,170.881,43.551,158.329
C01458=1034.934,257.481,-114.564,170.884,43.552,158.330
C01459=1034.940,257.729,-114.593,170.888,43.552,158.330
C01460=1034.947,257.977,-114.623,170.891,43.553,158.331
C01461=1034.954,258.225,-114.652,170.894,43.554,158.331
C01462=1034.961,258.473,-114.682,170.897,43.554,158.331
C01463=1034.968,258.722,-114.712,170.900,43.554,158.332
C01464=1034.974,258.970,-114.741,170.904,43.554,158.332
C01465=1034.981,259.218,-114.771,170.907,43.555,158.332
C01466=1034.988,259.466,-114.800,170.910,43.556,158.333
C01467=1034.995,259.714,-114.830,170.914,43.556,158.333
C01468=1035.002,259.962,-114.859,170.916,43.557,158.333
C01469=1035.009,260.210,-114.889,170.919,43.557,158.334
C01470=1035.016,260.459,-114.919,170.923,43.558,158.334
C01471=1035.022,260.707,-114.948,170.926,43.558,158.335
C01472=1035.029,260.955,-114.978,170.930,43.558,158.335
C01473=1035.036,261.203,-115.008,170.933,43.559,158.335
C01474=1035.044,261.451,-115.037,170.937,43.560,158.336
C01475=1035.050,261.699,-115.068,170.940,43.560,158.336
C01476=1035.056,261.947,-115.097,170.943,43.560,158.336
C01477=1035.063,262.196,-115.127,170.946,43.561,158.337
C01478=1035.070,262.443,-115.157,170.949,43.562,158.337
C01479=1035.079,262.780,-115.198,170.954,43.562,158.338
C01480=1035.087,263.115,-115.238,170.959,43.564,158.338
C01481=1035.097,263.452,-115.279,170.963,43.564,158.339
C01482=1035.106,263.788,-115.320,170.968,43.565,158.339
C01483=1035.113,264.036,-115.350,170.971,43.565,158.340
C01484=1035.119,264.283,-115.380,170.974,43.566,158.340
C01485=1035.126,264.532,-115.410,170.977,43.567,158.341
C01486=1035.133,264.780,-115.440,170.980,43.567,158.341
C01487=1035.139,265.027,-115.470,170.984,43.568,158.342
C01488=1035.147,265.276,-115.500,170.987,43.568,158.342
C01489=1035.153,265.524,-115.531,170.991,43.569,158.342
C01490=1035.160,265.772,-115.561,170.994,43.570,158.343
C01491=1035.167,266.020,-115.591,170.998,43.570,158.343
C01492=1035.173,266.268,-115.622,171.001,43.571,158.344
C01493=1035.180,266.516,-115.651,171.005,43.572,158.344
C01494=1035.187,266.764,-115.681,171.008,43.572,158.344
C01495=1035.193,267.013,-115.712,171.011,43.573,158.345
C01496=1035.200,267.260,-115.742,171.014,43.573,158.345
C01497=1035.207,267.508,-115.772,171.017,43.574,158.346
C01498=1035.213,267.757,-115.803,171.021,43.575,158.346
C01499=1035.221,268.005,-115.833,171.024,43.575,158.346
C01500=1035.226,268.253,-115.863,171.028,43.576,158.347
C01501=1035.234,268.501,-115.893,171.031,43.577,158.347
C01502=1035.241,268.749,-115.924,171.035,43.577,158.348
C01503=1035.247,268.997,-115.955,171.038,43.578,158.348
C01504=1035.254,269.245,-115.985,171.042,43.579,158.349
C01505=1035.260,269.493,-116.015,171.045,43.579,158.349
C01506=1035.268,269.742,-116.045,171.049,43.580,158.349
C01507=1035.274,269.989,-116.077,171.052,43.581,158.350
C01508=1035.281,270.237,-116.107,171.056,43.581,158.350
C01509=1035.287,270.486,-116.137,171.059,43.582,158.351
C01510=1035.294,270.734,-116.168,171.062,43.583,158.351
C01511=1035.301,270.981,-116.199,171.066,43.583,158.352
C01512=1035.308,271.229,-116.229,171.069,43.584,158.352
C01513=1035.314,271.478,-116.259,171.072,43.585,158.352
C01514=1035.322,271.725,-116.290,171.075,43.586,158.353
C01515=1035.328,271.974,-116.321,171.079,43.586,158.353
C01516=1035.334,272.222,-116.351,171.082,43.587,158.354
C01517=1035.341,272.469,-116.382,171.086,43.588,158.354
C01518=1035.348,272.718,-116.413,171.089,43.588,158.355
C01519=1035.355,272.965,-116.444,171.093,43.589,158.355
C01520=1035.362,273.214,-116.474,171.096,43.590,158.356
C01521=1035.367,273.462,-116.505,171.100,43.591,158.356
C01522=1035.375,273.709,-116.536,171.103,43.592,158.357
C01523=1035.381,273.958,-116.566,171.107,43.592,158.357
C01524=1035.389,274.205,-116.597,171.110,43.593,158.357
C01525=1035.395,274.454,-116.628,171.114,43.594,158.358
C01526=1035.402,274.702,-116.659,171.117,43.594,158.358
C01527=1035.408,274.950,-116.690,171.121,43.595,158.359
C01528=1035.415,275.197,-116.721,171.124,43.596,158.359
C01529=1035.422,275.445,-116.752,171.128,43.597,158.360
C01530=1035.428,275.694,-116.783,171.132,43.598,158.360
C01531=1035.436,275.941,-116.814,171.135,43.598,158.361
C01532=1035.442,276.190,-116.844,171.139,43.599,158.361
C01533=1035.449,276.438,-116.876,171.142,43.600,158.362
C01534=1035.456,276.685,-116.906,171.145,43.600,158.362
C01535=1035.465,277.026,-116.948,171.151,43.601,158.363
C01536=1035.475,277.366,-116.991,171.156,43.602,158.363
C01537=1035.484,277.707,-117.033,171.161,43.603,158.364
C01538=1035.493,278.048,-117.076,171.165,43.605,158.365
C01539=1035.500,278.295,-117.108,171.169,43.606,158.365
C01540=1035.506,278.544,-117.139,171.173,43.606,158.366
C01541=1035.513,278.792,-117.170,171.176,43.607,158.366
C01542=1035.520,279.040,-117.201,171.180,43.608,158.367
C01543=1035.527,279.288,-117.233,171.183,43.609,158.367
C01544=1035.533,279.536,-117.264,171.187,43.610,158.367
C01545=1035.540,279.784,-117.296,171.190,43.611,158.368
C01546=1035.547,280.031,-117.327,171.195,43.612,158.369
C01547=1035.553,280.279,-117.357,171.198,43.612,158.369
C01548=1035.559,280.527,-117.389,171.202,43.614,158.370
C01549=1035.566,280.775,-117.420,171.206,43.614,158.370
C01550=1035.573,281.023,-117.452,171.209,43.615,158.370
C01551=1035.580,281.271,-117.483,171.213,43.616,158.371
C01552=1035.587,281.518,-117.514,171.216,43.617,158.371
C01553=1035.594,281.766,-117.545,171.220,43.617,158.372
C01554=1035.600,282.014,-117.577,171.223,43.619,158.373
C01555=1035.607,282.262,-117.608,171.227,43.619,158.373
C01556=1035.614,282.510,-117.640,171.231,43.621,158.374
C01557=1035.621,282.758,-117.671,171.234,43.621,158.374
C01558=1035.628,283.007,-117.703,171.239,43.622,158.374
C01559=1035.635,283.254,-117.734,171.242,43.623,158.375
C01560=1035.641,283.502,-117.766,171.246,43.624,158.375
C01561=1035.648,283.750,-117.797,171.250,43.625,158.376
C01562=1035.655,283.998,-117.829,171.253,43.626,158.377
C01563=1035.661,284.246,-117.860,171.256,43.626,158.377
C01564=1035.669,284.493,-117.892,171.260,43.628,158.378
C01565=1035.675,284.741,-117.924,171.264,43.628,158.378
C01566=1035.682,284.989,-117.955,171.268,43.629,158.379
C01567=1035.689,285.237,-117.987,171.272,43.630,158.379
C01568=1035.695,285.485,-118.018,171.276,43.631,158.380
C01569=1035.703,285.734,-118.050,171.279,43.632,158.380
C01570=1035.709,285.981,-118.081,171.283,43.633,158.381
C01571=1035.716,286.229,-118.113,171.286,43.634,158.381
C01572=1035.723,286.477,-118.145,171.291,43.634,158.382
C01573=1035.730,286.725,-118.176,171.294,43.636,158.382
C01574=1035.737,286.972,-118.208,171.298,43.637,158.383
C01575=1035.744,287.220,-118.240,171.302,43.638,158.383
C01576=1035.750,287.468,-118.272,171.305,43.639,158.384
C01577=1035.757,287.717,-118.304,171.309,43.640,158.384
C01578=1035.764,287.964,-118.336,171.314,43.641,158.385
C01579=1035.771,288.212,-118.367,171.317,43.641,158.385
C01580=1035.778,288.459,-118.399,171.321,43.643,158.386
C01581=1035.785,288.707,-118.431,171.324,43.644,158.387
C01582=1035.791,288.956,-118.463,171.328,43.645,158.387
C01583=1035.798,289.203,-118.495,171.332,43.646,158.388
C01584=1035.805,289.451,-118.527,171.336,43.647,158.388
C01585=1035.812,289.698,-118.559,171.340,43.648,158.389
C01586=1035.818,289.947,-118.591,171.344,43.649,158.389
C01587=1035.825,290.194,-118.623,171.347,43.650,158.390
C01588=1035.832,290.442,-118.655,171.351,43.651,158.390
C01589=1035.839,290.690,-118.687,171.355,43.652,158.391
C01590=1035.845,290.938,-118.719,171.359,43.653,158.391
C01591=1035.856,291.290,-118.765,171.364,43.654,158.392
C01592=1035.865,291.643,-118.810,171.370,43.656,158.393
C01593=1035.875,291.996,-118.857,171.376,43.657,158.394
C01594=1035.884,292.348,-118.902,171.381,43.659,158.395
C01595=1035.892,292.596,-118.934,171.384,43.660,158.395
C01596=1035.898,292.843,-118.967,171.389,43.661,158.396
C01597=1035.905,293.091,-118.999,171.393,43.662,158.396
C01598=1035.913,293.339,-119.031,171.396,43.663,158.397
C01599=1035.919,293.587,-119.064,171.400,43.665,158.397
C01600=1035.926,293.835,-119.095,171.405,43.666,158.398
C01601=1035.933,294.083,-119.128,171.408,43.666,158.399
C01602=1035.940,294.330,-119.161,171.412,43.668,158.399
C01603=1035.947,294.578,-119.193,171.416,43.669,158.400
C01604=1035.953,294.826,-119.226,171.420,43.670,158.400
C01605=1035.960,295.074,-119.257,171.424,43.671,158.401
C01606=1035.967,295.322,-119.290,171.428,43.672,158.402
C01607=1035.973,295.569,-119.323,171.432,43.674,158.402
C01608=1035.980,295.817,-119.355,171.436,43.675,158.403
C01609=1035.987,296.065,-119.388,171.440,43.676,158.403
C01610=1035.993,296.312,-119.421,171.444,43.677,158.404
C01611=1036.000,296.561,-119.454,171.447,43.679,158.405
C01612=1036.007,296.808,-119.486,171.452,43.680,158.405
C01613=1036.013,297.055,-119.519,171.456,43.681,158.406
C01614=1036.020,297.304,-119.552,171.460,43.682,158.406
C01615=1036.026,297.551,-119.585,171.463,43.684,158.407
C01616=1036.034,297.798,-119.617,171.468,43.685,158.408
C01617=1036.041,298.046,-119.651,171.472,43.686,158.408
C01618=1036.047,298.294,-119.683,171.475,43.687,158.409
C01619=1036.053,298.541,-119.716,171.480,43.688,158.409
C01620=1036.061,298.789,-119.749,171.484,43.689,158.410
C01621=1036.067,299.037,-119.781,171.488,43.691,158.411
C01622=1036.074,299.285,-119.814,171.491,43.692,158.411
C01623=1036.081,299.532,-119.848,171.496,43.693,158.412
C01624=1036.088,299.780,-119.880,171.500,43.694,158.413
C01625=1036.095,300.028,-119.913,171.504,43.696,158.413
C01626=1036.101,300.276,-119.946,171.508,43.697,158.414
C01627=1036.108,300.524,-119.979,171.512,43.699,158.415
C01628=1036.115,300.770,-120.012,171.516,43.700,158.415
C01629=1036.122,301.019,-120.045,171.521,43.701,158.416
C01630=1036.128,301.266,-120.078,171.524,43.702,158.416
C01631=1036.135,301.514,-120.111,171.528,43.703,158.417
C01632=1036.143,301.761,-120.144,171.533,43.704,158.418
C01633=1036.149,302.010,-120.177,171.536,43.706,158.418
C01634=1036.156,302.257,-120.210,171.541,43.707,158.419
C01635=1036.163,302.505,-120.243,171.545,43.709,158.420
C01636=1036.169,302.752,-120.276,171.549,43.710,158.420
C01637=1036.177,303.000,-120.309,171.554,43.711,158.421
C01638=1036.184,303.248,-120.342,171.557,43.712,158.421
C01639=1036.191,303.495,-120.376,171.561,43.714,158.422
C01640=1036.198,303.743,-120.409,171.566,43.715,158.423
C01641=1036.205,303.991,-120.441,171.570,43.716,158.423
C01642=1036.212,304.238,-120.475,171.574,43.718,158.424
C01643=1036.218,304.486,-120.508,171.578,43.719,158.425
C01644=1036.225,304.734,-120.541,171.582,43.721,158.425
C01645=1036.232,304.982,-120.575,171.587,43.722,158.426
C01646=1036.239,305.229,-120.607,171.591,43.723,158.427
C01647=1036.250,305.599,-120.658,171.597,43.725,158.428
C01648=1036.260,305.967,-120.707,171.604,43.727,158.429
C01649=1036.270,306.337,-120.757,171.610,43.729,158.430
C01650=1036.281,306.706,-120.807,171.616,43.731,158.431
C01651=1036.288,306.955,-120.840,171.620,43.732,158.431
C01652=1036.295,307.202,-120.873,171.625,43.733,158.432
C01653=1036.303,307.449,-120.906,171.629,43.735,158.433
C01654=1036.310,307.697,-120.939,171.633,43.736,158.433
C01655=1036.316,307.944,-120.973,171.637,43.738,158.434
C01656=1036.324,308.192,-121.007,171.642,43.739,158.435
C01657=1036.330,308.440,-121.040,171.646,43.741,158.435
C01658=1036.338,308.688,-121.074,171.651,43.742,158.436
C01659=1036.345,308.935,-121.106,171.654,43.743,158.437
C01660=1036.352,309.182,-121.140,171.659,43.745,158.437
C01661=1036.359,309.430,-121.174,171.663,43.746,158.438
C01662=1036.366,309.678,-121.207,171.668,43.747,158.439
C01663=1036.374,309.926,-121.241,171.672,43.749,158.439
C01664=1036.381,310.173,-121.274,171.677,43.750,158.440
C01665=1036.388,310.420,-121.308,171.680,43.752,158.441
C01666=1036.395,310.668,-121.342,171.685,43.753,158.442
C01667=1036.402,310.916,-121.375,171.689,43.755,158.442
C01668=1036.409,311.164,-121.409,171.694,43.756,158.443
C01669=1036.417,311.412,-121.442,171.698,43.757,158.444
C01670=1036.424,311.659,-121.476,171.703,43.759,158.444
C01671=1036.430,311.906,-121.510,171.706,43.760,158.445
C01672=1036.438,312.154,-121.543,171.711,43.762,158.446
C01673=1036.445,312.401,-121.578,171.715,43.764,158.447
C01674=1036.452,312.649,-121.612,171.720,43.765,158.447
C01675=1036.458,312.896,-121.646,171.724,43.767,158.448
C01676=1036.465,313.144,-121.680,171.729,43.768,158.449
C01677=1036.472,313.392,-121.714,171.733,43.770,158.449
C01678=1036.479,313.639,-121.749,171.738,43.771,158.450
C01679=1036.486,313.887,-121.783,171.741,43.773,158.451
C01680=1036.492,314.134,-121.817,171.746,43.775,158.452
C01681=1036.499,314.382,-121.851,171.750,43.777,158.452
C01682=1036.506,314.629,-121.885,171.755,43.778,158.453
C01683=1036.513,314.877,-121.920,171.760,43.779,158.454
C01684=1036.520,315.124,-121.954,171.764,43.781,158.455
C01685=1036.527,315.371,-121.988,171.769,43.783,158.455
C01686=1036.534,315.619,-122.023,171.773,43.785,158.456
C01687=1036.541,315.867,-122.057,171.778,43.786,158.457
C01688=1036.548,316.114,-122.092,171.782,43.788,158.458
C01689=1036.555,316.362,-122.125,171.787,43.789,158.458
C01690=1036.561,316.609,-122.160,171.791,43.791,158.459
C01691=1036.568,316.856,-122.194,171.796,43.793,158.460
C01692=1036.576,317.103,-122.229,171.800,43.795,158.461
C01693=1036.582,317.351,-122.263,171.804,43.796,158.462
C01694=1036.590,317.598,-122.298,171.809,43.798,158.462
C01695=1036.596,317.846,-122.332,171.813,43.800,158.463
C01696=1036.604,318.093,-122.367,171.818,43.802,158.464
C01697=1036.610,318.341,-122.401,171.823,43.803,158.465
C01698=1036.618,318.589,-122.435,171.827,43.805,158.466
C01699=1036.624,318.836,-122.470,171.832,43.806,158.466
C01700=1036.632,319.084,-122.505,171.836,43.808,158.467
C01701=1036.639,319.332,-122.539,171.841,43.810,158.468
C01702=1036.646,319.579,-122.574,171.846,43.811,158.469
C01703=1036.657,319.953,-122.626,171.852,43.814,158.470
C01704=1036.668,320.328,-122.679,171.860,43.817,158.471
C01705=1036.679,320.702,-122.731,171.866,43.820,158.472
C01706=1036.690,321.076,-122.783,171.874,43.822,158.473
C01707=1036.697,321.323,-122.818,171.878,43.824,158.474
C01708=1036.704,321.571,-122.852,171.883,43.826,158.475
C01709=1036.711,321.818,-122.887,171.888,43.827,158.476
C01710=1036.718,322.065,-122.922,171.893,43.829,158.477
C01711=1036.725,322.313,-122.957,171.897,43.831,158.477
C01712=1036.733,322.561,-122.991,171.902,43.832,158.478
C01713=1036.739,322.808,-123.026,171.907,43.834,158.479
C01714=1036.747,323.056,-123.061,171.911,43.836,158.480
C01715=1036.754,323.303,-123.096,171.916,43.838,158.481
C01716=1036.762,323.551,-123.131,171.921,43.840,158.482
C01717=1036.769,323.798,-123.166,171.926,43.841,158.482
C01718=1036.776,324.045,-123.200,171.930,43.843,158.483
C01719=1036.783,324.292,-123.236,171.935,43.845,158.484
C01720=1036.791,324.540,-123.271,171.940,43.847,158.485
C01721=1036.798,324.788,-123.306,171.944,43.849,158.486
C01722=1036.805,325.035,-123.340,171.949,43.850,158.486
C01723=1036.813,325.283,-123.376,171.954,43.852,158.487
C01724=1036.820,325.530,-123.410,171.959,43.854,158.488
C01725=1036.827,325.777,-123.445,171.964,43.856,158.489
C01726=1036.835,326.025,-123.480,171.968,43.858,158.490
C01727=1036.842,326.272,-123.515,171.973,43.859,158.491
C01728=1036.849,326.520,-123.551,171.978,43.861,158.491
C01729=1036.857,326.767,-123.585,171.983,43.863,158.492
C01730=1036.863,327.015,-123.621,171.987,43.865,158.493
C01731=1036.872,327.262,-123.656,171.992,43.867,158.494
C01732=1036.878,327.510,-123.691,171.997,43.869,158.495
C01733=1036.886,327.758,-123.726,172.002,43.871,158.496
C01734=1036.893,328.004,-123.761,172.007,43.872,158.497
C01735=1036.901,328.251,-123.796,172.012,43.875,158.497
C01736=1036.908,328.499,-123.831,172.016,43.876,158.498
C01737=1036.915,328.747,-123.867,172.021,43.879,158.499
C01738=1036.923,328.994,-123.903,172.026,43.880,158.500
C01739=1036.930,329.242,-123.938,172.032,43.882,158.501
C01740=1036.937,329.488,-123.974,172.037,43.884,158.502
C01741=1036.945,329.736,-124.009,172.041,43.886,158.503
C01742=1036.952,329.983,-124.045,172.046,43.889,158.504
C01743=1036.959,330.231,-124.080,172.051,43.890,158.505
C01744=1036.966,330.478,-124.116,172.056,43.893,158.505
C01745=1036.974,330.726,-124.151,172.061,43.894,158.506
C01746=1036.981,330.972,-124.187,172.066,43.896,158.507
C01747=1036.988,331.221,-124.223,172.070,43.899,158.508
C01748=1036.995,331.467,-124.259,172.075,43.900,158.509
C01749=1037.002,331.715,-124.294,172.081,43.903,158.510
C01750=1037.010,331.962,-124.330,172.086,43.905,158.511
C01751=1037.017,332.210,-124.366,172.091,43.907,158.512
C01752=1037.024,332.457,-124.401,172.096,43.909,158.513
C01753=1037.032,332.704,-124.438,172.101,43.911,158.514
C01754=1037.039,332.951,-124.473,172.105,43.913,158.515
C01755=1037.046,333.199,-124.509,172.110,43.915,158.515
C01756=1037.054,333.447,-124.545,172.116,43.917,158.516
C01757=1037.061,333.693,-124.581,172.121,43.919,158.517
C01758=1037.068,333.941,-124.616,172.126,43.922,158.518
C01759=1037.079,334.311,-124.670,172.134,43.925,158.520
C01760=1037.091,334.681,-124.724,172.141,43.928,158.521
C01761=1037.102,335.050,-124.777,172.149,43.931,158.522
C01762=1037.112,335.419,-124.831,172.156,43.935,158.524
C01763=1037.120,335.667,-124.868,172.161,43.937,158.525
C01764=1037.127,335.913,-124.903,172.167,43.939,158.526
C01765=1037.134,336.161,-124.940,172.172,43.941,158.527
C01766=1037.142,336.409,-124.976,172.177,43.943,158.528
C01767=1037.149,336.655,-125.012,172.182,43.946,158.529
C01768=1037.156,336.903,-125.049,172.187,43.948,158.530
C01769=1037.163,337.151,-125.085,172.193,43.950,158.531
C01770=1037.171,337.397,-125.122,172.198,43.952,158.532
C01771=1037.178,337.644,-125.158,172.203,43.954,158.533
C01772=1037.186,337.892,-125.194,172.208,43.957,158.534
C01773=1037.194,338.139,-125.231,172.213,43.959,158.535
C01774=1037.201,338.387,-125.267,172.219,43.961,158.536
C01775=1037.208,338.634,-125.303,172.224,43.963,158.537
C01776=1037.215,338.881,-125.339,172.229,43.965,158.538
C01777=1037.223,339.128,-125.376,172.235,43.968,158.539
C01778=1037.230,339.376,-125.413,172.240,43.971,158.540
C01779=1037.238,339.623,-125.449,172.245,43.973,158.541
C01780=1037.245,339.870,-125.485,172.250,43.975,158.542
C01781=1037.253,340.117,-125.522,172.255,43.977,158.543
C01782=1037.260,340.364,-125.559,172.261,43.980,158.544
C01783=1037.268,340.612,-125.595,172.266,43.982,158.545
C01784=1037.276,340.859,-125.632,172.271,43.984,158.546
C01785=1037.283,341.106,-125.668,172.277,43.987,158.547
C01786=1037.291,341.353,-125.706,172.282,43.989,158.548
C01787=1037.298,341.600,-125.742,172.287,43.991,158.549
C01788=1037.305,341.847,-125.779,172.292,43.994,158.550
C01789=1037.313,342.095,-125.816,172.298,43.996,158.551
C01790=1037.320,342.342,-125.853,172.303,43.999,158.552
C01791=1037.327,342.589,-125.889,172.309,44.001,158.553
C01792=1037.335,342.836,-125.927,172.315,44.003,158.554
C01793=1037.342,343.084,-125.963,172.320,44.006,158.555
C01794=1037.350,343.331,-126.001,172.325,44.008,158.556
C01795=1037.358,343.578,-126.037,172.331,44.011,158.557
C01796=1037.365,343.825,-126.074,172.336,44.013,158.558
C01797=1037.372,344.072,-126.111,172.341,44.016,158.559
C01798=1037.380,344.319,-126.149,172.347,44.018,158.561
